SPLINE
SPL {X  -134.058, Y  +288.094, Z    +0.000, E1   +46.503, E3 +198295.093}
SPL {X  -148.633, Y  +314.028, Z    +0.000, E1   +38.752, E3 +198303.982}
SPL {X  -156.325, Y  +334.971, Z    +0.000, E1   +30.037, E3 +198307.750}
SPL {X  -160.130, Y  +351.024, Z    +0.000, E1   +21.715, E3 +198311.064}
SPL {X  -162.127, Y  +365.491, Z    +0.000, E1   +12.692, E3 +198310.988}
SPL {X  -162.801, Y  +378.004, Z    +0.000, E1    +3.811, E3 +198311.404}
SPL {X  -162.820, Y  +382.501, Z    +0.000, E1    +0.028, E3 +198310.822}
SPL {X  -162.820, Y  +385.123, Z    +0.000, E1    -3.284, E3 +198310.499}
SPL {X  -162.820, Y  +390.608, Z    +0.000, E1   -12.198, E3 +198310.413}
SPL {X  -162.820, Y  +396.028, Z    +0.000, E1   -22.022, E3 +198310.281}
SPL {X  -162.820, Y  +402.037, Z    +0.000, E1   -32.247, E3 +198310.219}
SPL {X  -162.820, Y  +411.189, Z    +0.000, E1   -44.140, E3 +198311.548}
SPL {X  -162.820, Y  +422.160, Z    +0.000, E1   -56.042, E3 +198310.020}
SPL {X  -162.820, Y  +475.891, Z    +0.000, E1   -67.666, E3 +198330.339}
SPL {X  -162.820, Y  +573.811, Z    +0.000, E1   -65.269, E3 +198414.937}
SPL {X  -162.820, Y  +580.233, Z    +0.000, E1   -64.427, E3 +198427.644}
SPL {X  -162.820, Y  +590.756, Z    +0.000, E1   -64.410, E3 +198438.211}
SPL {X  -162.820, Y  +600.605, Z    +0.000, E1   -64.446, E3 +198447.785}
SPL {X  -162.820, Y  +611.699, Z    +0.000, E1   -64.369, E3 +198459.464}
SPL {X  -162.820, Y  +622.825, Z    +0.000, E1   -64.446, E3 +198469.909}
SPL {X  -162.820, Y  +635.776, Z    +0.000, E1   -64.495, E3 +198482.598}
SPL {X  -162.820, Y  +648.933, Z    +0.000, E1   -64.417, E3 +198496.145}
SPL {X  -162.820, Y  +658.800, Z    +0.000, E1   -64.418, E3 +198505.960}
SPL {X  -162.820, Y  +670.777, Z    +0.000, E1   -64.432, E3 +198517.873}
SPL {X  -162.296, Y  +686.556, Z    +0.000, E1   -64.388, E3 +198534.076}
SPL {X  -160.469, Y  +701.070, Z    +0.000, E1   -64.058, E3 +198550.979}
SPL {X  -157.811, Y  +713.575, Z    +0.000, E1   -63.758, E3 +198565.558}
SPL {X  -155.696, Y  +721.135, Z    +0.000, E1   -63.387, E3 +198575.491}
SPL {X  -153.915, Y  +726.609, Z    +0.000, E1   -63.196, E3 +198582.266}
SPL {X  -151.802, Y  +732.376, Z    +0.000, E1   -62.761, E3 +198590.807}
SPL {X  -149.758, Y  +737.398, Z    +0.000, E1   -62.434, E3 +198597.828}
SPL {X  -146.903, Y  +743.713, Z    +0.000, E1   -62.188, E3 +198605.600}
SPL {X  -143.515, Y  +750.401, Z    +0.000, E1   -61.484, E3 +198616.285}
SPL {X  -140.303, Y  +756.116, Z    +0.000, E1   -60.974, E3 +198624.482}
SPL {X  -137.988, Y  +759.927, Z    +0.000, E1   -60.537, E3 +198630.416}
SPL {X  -134.516, Y  +765.238, Z    +0.000, E1   -60.629, E3 +198635.219}
SPL {X  -126.113, Y  +776.485, Z    +0.000, E1   -62.672, E3 +198636.779}
SPL {X   -95.040, Y  +805.704, Z    +0.000, E1   -55.103, E3 +198727.739}
ENDSPLINE

SPLINE
SPL {X   -95.634, Y  +805.274, Z    +0.000, E1   -52.767, E3 +198766.898}
SPL {X  -130.051, Y  +771.465, Z    +0.000, E1   -46.832, E3 +198865.304}
SPL {X  -154.243, Y  +725.647, Z    +0.000, E1   -32.659, E3 +198886.866}
SPL {X  -160.324, Y  +701.901, Z    +0.000, E1   -20.534, E3 +198887.689}
SPL {X  -161.938, Y  +690.423, Z    +0.000, E1   -13.625, E3 +198889.080}
SPL {X  -162.746, Y  +678.392, Z    +0.000, E1    -5.513, E3 +198889.152}
SPL {X  -162.820, Y  +671.700, Z    +0.000, E1    -0.272, E3 +198888.718}
SPL {X  -162.820, Y  +668.888, Z    +0.000, E1    +3.063, E3 +198888.415}
SPL {X  -162.820, Y  +664.763, Z    +0.000, E1    +9.526, E3 +198888.075}
SPL {X  -162.820, Y  +660.761, Z    +0.000, E1   +16.102, E3 +198888.414}
SPL {X  -162.820, Y  +655.024, Z    +0.000, E1   +25.730, E3 +198888.575}
SPL {X  -162.820, Y  +646.498, Z    +0.000, E1   +39.738, E3 +198887.096}
SPL {X  -162.820, Y  +637.711, Z    +0.000, E1   +46.793, E3 +198891.589}
SPL {X  -162.820, Y  +598.602, Z    +0.000, E1   +67.541, E3 +198894.140}
SPL {X  -162.820, Y  +578.435, Z    +0.000, E1   +65.472, E3 +198912.240}
SPL {X  -162.820, Y  +475.450, Z    +0.000, E1   +67.130, E3 +198981.177}
ENDSPLINE

SPLINE
SPL {X  -162.820, Y  +483.223, Z    +0.000, E1   +64.312, E3 +198995.617}
SPL {X  -162.820, Y  +502.830, Z    +0.000, E1   +59.229, E3 +199010.538}
ENDSPLINE

SPLINE
SPL {X  -162.820, Y  +486.621, Z    +0.000, E1   +59.661, E3 +199027.457}
SPL {X  -162.820, Y  +472.771, Z    +0.000, E1   +60.369, E3 +199039.203}
SPL {X  -162.820, Y  +460.138, Z    +0.000, E1   +61.014, E3 +199049.522}
SPL {X  -162.820, Y  +448.741, Z    +0.000, E1   +61.510, E3 +199059.037}
SPL {X  -162.820, Y  +430.985, Z    +0.000, E1   +62.533, E3 +199071.470}
SPL {X  -162.820, Y  +413.005, Z    +0.000, E1   +63.234, E3 +199085.460}
SPL {X  -162.820, Y  +396.727, Z    +0.000, E1   +63.972, E3 +199096.811}
SPL {X  -162.756, Y  +375.937, Z    +0.000, E1   +64.914, E3 +199110.421}
SPL {X  -161.353, Y  +358.691, Z    +0.000, E1   +65.588, E3 +199121.645}
SPL {X  -158.833, Y  +344.688, Z    +0.000, E1   +65.800, E3 +199133.108}
SPL {X  -156.326, Y  +334.977, Z    +0.000, E1   +65.428, E3 +199144.581}
SPL {X  -153.776, Y  +326.991, Z    +0.000, E1   +65.023, E3 +199154.844}
SPL {X  -149.992, Y  +317.154, Z    +0.000, E1   +64.515, E3 +199167.308}
SPL {X  -146.026, Y  +308.480, Z    +0.000, E1   +63.813, E3 +199179.550}
SPL {X  -142.454, Y  +301.650, Z    +0.000, E1   +63.360, E3 +199188.314}
SPL {X  -139.696, Y  +296.861, Z    +0.000, E1   +62.910, E3 +199195.082}
SPL {X  -137.330, Y  +293.030, Z    +0.000, E1   +62.290, E3 +199201.706}
SPL {X  -134.245, Y  +288.366, Z    +0.000, E1   +62.031, E3 +199207.188}
SPL {X  -128.642, Y  +280.693, Z    +0.000, E1   +63.351, E3 +199208.181}
SPL {X   -90.696, Y  +245.280, Z    +0.000, E1   +54.124, E3 +199328.870}
ENDSPLINE

SPLINE
SPL {X  -134.058, Y  +288.094, Z    +0.000, E1   +46.503, E3 +199456.384}
SPL {X  -153.979, Y  +327.577, Z    +0.000, E1   +33.452, E3 +199467.924}
SPL {X  -160.130, Y  +351.024, Z    +0.000, E1   +21.715, E3 +199472.354}
SPL {X  -162.127, Y  +365.491, Z    +0.000, E1   +12.692, E3 +199472.278}
SPL {X  -162.801, Y  +378.004, Z    +0.000, E1    +3.811, E3 +199472.694}
SPL {X  -162.820, Y  +382.501, Z    +0.000, E1    +0.028, E3 +199472.112}
SPL {X  -162.820, Y  +385.123, Z    +0.000, E1    -3.284, E3 +199471.790}
SPL {X  -162.820, Y  +390.608, Z    +0.000, E1   -12.198, E3 +199471.703}
SPL {X  -162.820, Y  +396.028, Z    +0.000, E1   -22.022, E3 +199471.571}
SPL {X  -162.820, Y  +402.037, Z    +0.000, E1   -32.247, E3 +199471.509}
SPL {X  -162.820, Y  +414.067, Z    +0.000, E1   -47.235, E3 +199472.935}
SPL {X  -162.820, Y  +424.566, Z    +0.000, E1   -59.255, E3 +199469.600}
SPL {X  -162.820, Y  +460.664, Z    +0.000, E1   -69.605, E3 +199477.896}
SPL {X  -162.820, Y  +481.040, Z    +0.000, E1   -67.047, E3 +199496.485}
SPL {X  -162.820, Y  +576.352, Z    +0.000, E1   -67.140, E3 +199564.004}
ENDSPLINE

SPLINE
SPL {X  -162.820, Y  +573.336, Z    +0.000, E1   -64.995, E3 +199577.756}
ENDSPLINE

SPLINE
SPL {X  -162.820, Y  +580.233, Z    +0.000, E1   -64.427, E3 +199588.934}
SPL {X  -162.820, Y  +590.756, Z    +0.000, E1   -64.410, E3 +199599.502}
SPL {X  -162.820, Y  +600.605, Z    +0.000, E1   -64.446, E3 +199609.075}
SPL {X  -162.820, Y  +611.699, Z    +0.000, E1   -64.369, E3 +199620.754}
SPL {X  -162.820, Y  +622.825, Z    +0.000, E1   -64.446, E3 +199631.199}
SPL {X  -162.820, Y  +635.776, Z    +0.000, E1   -64.495, E3 +199643.889}
SPL {X  -162.820, Y  +648.933, Z    +0.000, E1   -64.417, E3 +199657.436}
SPL {X  -162.820, Y  +658.800, Z    +0.000, E1   -64.418, E3 +199667.250}
SPL {X  -162.820, Y  +670.777, Z    +0.000, E1   -64.432, E3 +199679.163}
SPL {X  -162.296, Y  +686.556, Z    +0.000, E1   -64.388, E3 +199695.366}
SPL {X  -160.469, Y  +701.070, Z    +0.000, E1   -64.058, E3 +199712.269}
SPL {X  -157.811, Y  +713.575, Z    +0.000, E1   -63.758, E3 +199726.848}
SPL {X  -154.601, Y  +724.576, Z    +0.000, E1   -63.303, E3 +199740.970}
SPL {X  -151.802, Y  +732.376, Z    +0.000, E1   -62.761, E3 +199752.097}
SPL {X  -149.758, Y  +737.398, Z    +0.000, E1   -62.434, E3 +199759.118}
SPL {X  -146.903, Y  +743.713, Z    +0.000, E1   -62.188, E3 +199766.891}
SPL {X  -143.515, Y  +750.401, Z    +0.000, E1   -61.484, E3 +199777.575}
SPL {X  -138.985, Y  +758.314, Z    +0.000, E1   -60.770, E3 +199789.134}
SPL {X  -133.449, Y  +766.783, Z    +0.000, E1   -60.899, E3 +199796.754}
SPL {X   -94.739, Y  +805.919, Z    +0.000, E1   -54.063, E3 +199904.811}
ENDSPLINE

SPLINE
SPL {X  -130.051, Y  +771.465, Z    +0.000, E1   -46.832, E3 +200026.595}
SPL {X  -154.243, Y  +725.647, Z    +0.000, E1   -32.659, E3 +200048.157}
SPL {X  -160.324, Y  +701.901, Z    +0.000, E1   -20.534, E3 +200048.980}
SPL {X  -161.938, Y  +690.423, Z    +0.000, E1   -13.625, E3 +200050.370}
SPL {X  -162.638, Y  +681.194, Z    +0.000, E1    -7.430, E3 +200050.191}
SPL {X  -162.820, Y  +672.793, Z    +0.000, E1    -1.263, E3 +200050.249}
SPL {X  -162.820, Y  +670.674, Z    +0.000, E1    +0.808, E3 +200049.779}
SPL {X  -162.820, Y  +666.307, Z    +0.000, E1    +6.851, E3 +200049.562}
SPL {X  -162.820, Y  +660.761, Z    +0.000, E1   +16.102, E3 +200049.705}
SPL {X  -162.820, Y  +655.024, Z    +0.000, E1   +25.730, E3 +200049.866}
SPL {X  -162.820, Y  +646.498, Z    +0.000, E1   +39.738, E3 +200048.387}
SPL {X  -162.820, Y  +637.711, Z    +0.000, E1   +46.793, E3 +200052.879}
SPL {X  -162.820, Y  +598.602, Z    +0.000, E1   +67.541, E3 +200055.430}
SPL {X  -162.820, Y  +578.435, Z    +0.000, E1   +65.472, E3 +200073.530}
SPL {X  -162.820, Y  +480.401, Z    +0.000, E1   +65.660, E3 +200149.459}
ENDSPLINE

SPLINE
SPL {X  -162.820, Y  +490.253, Z    +0.000, E1   +62.754, E3 +200161.222}
SPL {X  -162.820, Y  +503.236, Z    +0.000, E1   +58.858, E3 +200173.575}
ENDSPLINE

SPLINE
SPL {X  -162.820, Y  +486.621, Z    +0.000, E1   +59.661, E3 +200188.748}
SPL {X  -162.820, Y  +472.771, Z    +0.000, E1   +60.369, E3 +200200.493}
SPL {X  -162.820, Y  +460.138, Z    +0.000, E1   +61.014, E3 +200210.813}
SPL {X  -162.820, Y  +448.741, Z    +0.000, E1   +61.510, E3 +200220.327}
SPL {X  -162.820, Y  +430.985, Z    +0.000, E1   +62.533, E3 +200232.760}
SPL {X  -162.820, Y  +413.005, Z    +0.000, E1   +63.234, E3 +200246.750}
SPL {X  -162.820, Y  +396.727, Z    +0.000, E1   +63.972, E3 +200258.102}
SPL {X  -162.756, Y  +375.937, Z    +0.000, E1   +64.914, E3 +200271.711}
SPL {X  -161.353, Y  +358.691, Z    +0.000, E1   +65.588, E3 +200282.936}
SPL {X  -159.475, Y  +347.667, Z    +0.000, E1   +65.889, E3 +200290.816}
SPL {X  -157.043, Y  +337.513, Z    +0.000, E1   +65.541, E3 +200302.894}
SPL {X  -154.736, Y  +329.832, Z    +0.000, E1   +65.034, E3 +200313.340}
SPL {X  -151.631, Y  +321.184, Z    +0.000, E1   +64.776, E3 +200323.185}
SPL {X  -147.832, Y  +312.265, Z    +0.000, E1   +64.201, E3 +200334.994}
SPL {X  -145.264, Y  +306.955, Z    +0.000, E1   +63.555, E3 +200343.600}
SPL {X  -142.454, Y  +301.650, Z    +0.000, E1   +63.360, E3 +200349.604}
SPL {X  -139.696, Y  +296.861, Z    +0.000, E1   +62.910, E3 +200356.372}
SPL {X  -137.330, Y  +293.030, Z    +0.000, E1   +62.290, E3 +200362.997}
SPL {X  -134.245, Y  +288.366, Z    +0.000, E1   +62.031, E3 +200368.478}
SPL {X  -128.642, Y  +280.693, Z    +0.000, E1   +63.351, E3 +200369.472}
SPL {X   -90.696, Y  +245.280, Z    +0.000, E1   +54.124, E3 +200490.160}
ENDSPLINE

SPLINE
SPL {X  -134.058, Y  +288.094, Z    +0.000, E1   +46.503, E3 +200617.674}
SPL {X  -153.979, Y  +327.577, Z    +0.000, E1   +33.452, E3 +200629.214}
SPL {X  -160.130, Y  +351.024, Z    +0.000, E1   +21.715, E3 +200633.645}
SPL {X  -162.127, Y  +365.491, Z    +0.000, E1   +12.692, E3 +200633.568}
SPL {X  -162.745, Y  +375.564, Z    +0.000, E1    +5.577, E3 +200634.179}
SPL {X  -162.820, Y  +382.222, Z    +0.000, E1    +0.380, E3 +200633.451}
SPL {X  -162.820, Y  +384.010, Z    +0.000, E1    -1.878, E3 +200633.114}
SPL {X  -162.820, Y  +387.631, Z    +0.000, E1    -7.169, E3 +200633.067}
SPL {X  -162.820, Y  +394.064, Z    +0.000, E1   -18.298, E3 +200632.878}
SPL {X  -162.820, Y  +402.037, Z    +0.000, E1   -32.247, E3 +200632.799}
SPL {X  -162.820, Y  +411.189, Z    +0.000, E1   -44.140, E3 +200634.129}
SPL {X  -162.820, Y  +422.160, Z    +0.000, E1   -56.042, E3 +200632.601}
SPL {X  -162.820, Y  +475.891, Z    +0.000, E1   -67.666, E3 +200652.919}
SPL {X  -162.820, Y  +573.811, Z    +0.000, E1   -65.269, E3 +200737.518}
SPL {X  -162.820, Y  +580.233, Z    +0.000, E1   -64.427, E3 +200750.224}
SPL {X  -162.820, Y  +590.756, Z    +0.000, E1   -64.410, E3 +200760.792}
SPL {X  -162.820, Y  +600.605, Z    +0.000, E1   -64.446, E3 +200770.365}
SPL {X  -162.820, Y  +611.699, Z    +0.000, E1   -64.369, E3 +200782.045}
SPL {X  -162.820, Y  +622.825, Z    +0.000, E1   -64.446, E3 +200792.489}
SPL {X  -162.820, Y  +635.776, Z    +0.000, E1   -64.495, E3 +200805.179}
SPL {X  -162.820, Y  +648.933, Z    +0.000, E1   -64.417, E3 +200818.726}
SPL {X  -162.820, Y  +658.800, Z    +0.000, E1   -64.418, E3 +200828.540}
SPL {X  -162.820, Y  +670.777, Z    +0.000, E1   -64.432, E3 +200840.453}
SPL {X  -162.296, Y  +686.556, Z    +0.000, E1   -64.388, E3 +200856.657}
SPL {X  -160.469, Y  +701.070, Z    +0.000, E1   -64.058, E3 +200873.560}
SPL {X  -157.811, Y  +713.575, Z    +0.000, E1   -63.758, E3 +200888.138}
SPL {X  -155.696, Y  +721.135, Z    +0.000, E1   -63.387, E3 +200898.072}
SPL {X  -153.915, Y  +726.609, Z    +0.000, E1   -63.196, E3 +200904.846}
SPL {X  -151.802, Y  +732.376, Z    +0.000, E1   -62.761, E3 +200913.388}
SPL {X  -149.758, Y  +737.398, Z    +0.000, E1   -62.434, E3 +200920.408}
SPL {X  -146.903, Y  +743.713, Z    +0.000, E1   -62.188, E3 +200928.181}
SPL {X  -144.901, Y  +747.758, Z    +0.000, E1   -61.566, E3 +200935.644}
SPL {X  -141.375, Y  +754.268, Z    +0.000, E1   -61.208, E3 +200944.198}
SPL {X  -137.124, Y  +761.291, Z    +0.000, E1   -60.398, E3 +200955.109}
SPL {X  -130.896, Y  +770.333, Z    +0.000, E1   -61.755, E3 +200957.784}
SPL {X   -94.739, Y  +805.919, Z    +0.000, E1   -54.063, E3 +201066.101}
ENDSPLINE

SPLINE
SPL {X  -130.051, Y  +771.465, Z    +0.000, E1   -46.832, E3 +201187.885}
SPL {X  -150.288, Y  +736.141, Z    +0.000, E1   -36.889, E3 +201207.741}
SPL {X  -159.122, Y  +708.003, Z    +0.000, E1   -24.018, E3 +201210.449}
SPL {X  -161.938, Y  +690.423, Z    +0.000, E1   -13.625, E3 +201211.660}
SPL {X  -162.746, Y  +678.392, Z    +0.000, E1    -5.513, E3 +201211.733}
SPL {X  -162.820, Y  +671.700, Z    +0.000, E1    -0.272, E3 +201211.299}
SPL {X  -162.820, Y  +668.888, Z    +0.000, E1    +3.063, E3 +201210.996}
SPL {X  -162.820, Y  +664.763, Z    +0.000, E1    +9.526, E3 +201210.655}
SPL {X  -162.820, Y  +660.761, Z    +0.000, E1   +16.102, E3 +201210.995}
SPL {X  -162.820, Y  +655.024, Z    +0.000, E1   +25.730, E3 +201211.156}
SPL {X  -162.820, Y  +646.498, Z    +0.000, E1   +39.738, E3 +201209.677}
SPL {X  -162.820, Y  +637.711, Z    +0.000, E1   +46.793, E3 +201214.170}
SPL {X  -162.820, Y  +613.264, Z    +0.000, E1   +68.325, E3 +201206.368}
SPL {X  -162.820, Y  +583.199, Z    +0.000, E1   +66.160, E3 +201229.858}
SPL {X  -162.820, Y  +480.401, Z    +0.000, E1   +65.660, E3 +201310.749}
ENDSPLINE

SPLINE
SPL {X  -162.820, Y  +490.253, Z    +0.000, E1   +62.754, E3 +201322.512}
SPL {X  -162.820, Y  +503.236, Z    +0.000, E1   +58.858, E3 +201334.866}
ENDSPLINE

SPLINE
SPL {X  -162.820, Y  +486.621, Z    +0.000, E1   +59.661, E3 +201350.038}
SPL {X  -162.820, Y  +472.771, Z    +0.000, E1   +60.369, E3 +201361.783}
SPL {X  -162.820, Y  +460.138, Z    +0.000, E1   +61.014, E3 +201372.103}
SPL {X  -162.820, Y  +448.741, Z    +0.000, E1   +61.510, E3 +201381.618}
SPL {X  -162.820, Y  +430.985, Z    +0.000, E1   +62.533, E3 +201394.051}
SPL {X  -162.820, Y  +413.005, Z    +0.000, E1   +63.234, E3 +201408.041}
SPL {X  -162.820, Y  +396.727, Z    +0.000, E1   +63.972, E3 +201419.392}
SPL {X  -162.756, Y  +375.937, Z    +0.000, E1   +64.914, E3 +201433.001}
SPL {X  -161.353, Y  +358.691, Z    +0.000, E1   +65.588, E3 +201444.226}
SPL {X  -159.475, Y  +347.667, Z    +0.000, E1   +65.889, E3 +201452.107}
SPL {X  -157.043, Y  +337.513, Z    +0.000, E1   +65.541, E3 +201464.184}
SPL {X  -153.776, Y  +326.991, Z    +0.000, E1   +65.023, E3 +201477.425}
SPL {X  -149.992, Y  +317.154, Z    +0.000, E1   +64.515, E3 +201489.889}
SPL {X  -146.026, Y  +308.480, Z    +0.000, E1   +63.813, E3 +201502.131}
SPL {X  -142.454, Y  +301.650, Z    +0.000, E1   +63.360, E3 +201510.894}
SPL {X  -139.696, Y  +296.861, Z    +0.000, E1   +62.910, E3 +201517.662}
SPL {X  -137.330, Y  +293.030, Z    +0.000, E1   +62.290, E3 +201524.287}
SPL {X  -134.245, Y  +288.366, Z    +0.000, E1   +62.031, E3 +201529.769}
SPL {X  -128.642, Y  +280.693, Z    +0.000, E1   +63.351, E3 +201530.762}
SPL {X   -90.696, Y  +245.280, Z    +0.000, E1   +54.124, E3 +201651.451}
ENDSPLINE

SPLINE
SPL {X  -134.058, Y  +288.094, Z    +0.000, E1   +46.503, E3 +201778.964}
SPL {X  -153.979, Y  +327.577, Z    +0.000, E1   +33.452, E3 +201790.504}
SPL {X  -160.130, Y  +351.024, Z    +0.000, E1   +21.715, E3 +201794.935}
SPL {X  -162.127, Y  +365.491, Z    +0.000, E1   +12.692, E3 +201794.859}
SPL {X  -162.745, Y  +375.564, Z    +0.000, E1    +5.577, E3 +201795.469}
SPL {X  -162.820, Y  +382.222, Z    +0.000, E1    +0.380, E3 +201794.742}
SPL {X  -162.820, Y  +385.123, Z    +0.000, E1    -3.284, E3 +201794.370}
SPL {X  -162.820, Y  +390.608, Z    +0.000, E1   -12.198, E3 +201794.284}
SPL {X  -162.820, Y  +396.028, Z    +0.000, E1   -22.022, E3 +201794.152}
SPL {X  -162.820, Y  +402.037, Z    +0.000, E1   -32.247, E3 +201794.090}
SPL {X  -162.820, Y  +411.189, Z    +0.000, E1   -44.140, E3 +201795.419}
SPL {X  -162.820, Y  +422.160, Z    +0.000, E1   -56.042, E3 +201793.891}
SPL {X  -162.820, Y  +475.891, Z    +0.000, E1   -67.666, E3 +201814.210}
SPL {X  -162.820, Y  +573.811, Z    +0.000, E1   -65.269, E3 +201898.808}
SPL {X  -162.820, Y  +580.233, Z    +0.000, E1   -64.427, E3 +201911.515}
SPL {X  -162.820, Y  +590.756, Z    +0.000, E1   -64.410, E3 +201922.082}
SPL {X  -162.820, Y  +600.605, Z    +0.000, E1   -64.446, E3 +201931.656}
SPL {X  -162.820, Y  +611.699, Z    +0.000, E1   -64.369, E3 +201943.335}
SPL {X  -162.820, Y  +622.825, Z    +0.000, E1   -64.446, E3 +201953.780}
SPL {X  -162.820, Y  +635.776, Z    +0.000, E1   -64.495, E3 +201966.469}
SPL {X  -162.820, Y  +648.933, Z    +0.000, E1   -64.417, E3 +201980.016}
SPL {X  -162.820, Y  +658.800, Z    +0.000, E1   -64.418, E3 +201989.831}
SPL {X  -162.820, Y  +670.777, Z    +0.000, E1   -64.432, E3 +202001.744}
SPL {X  -162.296, Y  +686.556, Z    +0.000, E1   -64.388, E3 +202017.947}
SPL {X  -160.469, Y  +701.070, Z    +0.000, E1   -64.058, E3 +202034.850}
SPL {X  -157.811, Y  +713.575, Z    +0.000, E1   -63.758, E3 +202049.429}
SPL {X  -155.696, Y  +721.135, Z    +0.000, E1   -63.387, E3 +202059.362}
SPL {X  -153.915, Y  +726.609, Z    +0.000, E1   -63.196, E3 +202066.137}
SPL {X  -151.802, Y  +732.376, Z    +0.000, E1   -62.761, E3 +202074.678}
SPL {X  -149.758, Y  +737.398, Z    +0.000, E1   -62.434, E3 +202081.699}
SPL {X  -146.903, Y  +743.713, Z    +0.000, E1   -62.188, E3 +202089.471}
SPL {X  -143.515, Y  +750.401, Z    +0.000, E1   -61.484, E3 +202100.156}
SPL {X  -140.303, Y  +756.116, Z    +0.000, E1   -60.974, E3 +202108.353}
SPL {X  -137.124, Y  +761.291, Z    +0.000, E1   -60.398, E3 +202116.400}
SPL {X  -130.896, Y  +770.333, Z    +0.000, E1   -61.755, E3 +202119.074}
SPL {X   -94.739, Y  +805.919, Z    +0.000, E1   -54.063, E3 +202227.391}
ENDSPLINE

SPLINE
SPL {X  -130.051, Y  +771.465, Z    +0.000, E1   -46.832, E3 +202349.175}
SPL {X  -154.243, Y  +725.647, Z    +0.000, E1   -32.659, E3 +202370.737}
SPL {X  -161.394, Y  +695.005, Z    +0.000, E1   -16.571, E3 +202372.442}
SPL {X  -162.746, Y  +678.392, Z    +0.000, E1    -5.513, E3 +202373.023}
SPL {X  -162.820, Y  +672.097, Z    +0.000, E1    -0.584, E3 +202372.728}
SPL {X  -162.820, Y  +671.335, Z    +0.000, E1    +0.161, E3 +202372.461}
SPL {X  -162.820, Y  +668.888, Z    +0.000, E1    +3.063, E3 +202372.286}
SPL {X  -162.820, Y  +664.763, Z    +0.000, E1    +9.526, E3 +202371.946}
SPL {X  -162.820, Y  +660.761, Z    +0.000, E1   +16.102, E3 +202372.285}
SPL {X  -162.820, Y  +655.024, Z    +0.000, E1   +25.730, E3 +202372.446}
SPL {X  -162.820, Y  +646.498, Z    +0.000, E1   +39.738, E3 +202370.967}
SPL {X  -162.820, Y  +637.711, Z    +0.000, E1   +46.793, E3 +202375.460}
SPL {X  -162.820, Y  +598.602, Z    +0.000, E1   +67.541, E3 +202378.011}
SPL {X  -162.820, Y  +578.435, Z    +0.000, E1   +65.472, E3 +202396.111}
SPL {X  -162.820, Y  +480.401, Z    +0.000, E1   +65.660, E3 +202472.040}
ENDSPLINE

SPLINE
SPL {X  -162.820, Y  +490.253, Z    +0.000, E1   +62.754, E3 +202483.802}
SPL {X  -162.820, Y  +503.236, Z    +0.000, E1   +58.858, E3 +202496.156}
ENDSPLINE

SPLINE
SPL {X  -162.820, Y  +486.621, Z    +0.000, E1   +59.661, E3 +202511.328}
SPL {X  -162.820, Y  +472.771, Z    +0.000, E1   +60.369, E3 +202523.074}
SPL {X  -162.820, Y  +460.138, Z    +0.000, E1   +61.014, E3 +202533.393}
SPL {X  -162.820, Y  +442.137, Z    +0.000, E1   +61.946, E3 +202547.290}
SPL {X  -162.820, Y  +425.982, Z    +0.000, E1   +62.713, E3 +202559.316}
SPL {X  -162.820, Y  +413.005, Z    +0.000, E1   +63.234, E3 +202569.331}
SPL {X  -162.820, Y  +396.727, Z    +0.000, E1   +63.972, E3 +202580.682}
SPL {X  -162.820, Y  +382.966, Z    +0.000, E1   +64.511, E3 +202590.405}
SPL {X  -161.867, Y  +362.911, Z    +0.000, E1   +65.480, E3 +202602.478}
SPL {X  -158.833, Y  +344.688, Z    +0.000, E1   +65.800, E3 +202616.979}
SPL {X  -156.326, Y  +334.977, Z    +0.000, E1   +65.428, E3 +202628.452}
SPL {X  -153.776, Y  +326.991, Z    +0.000, E1   +65.023, E3 +202638.715}
SPL {X  -150.991, Y  +319.573, Z    +0.000, E1   +64.614, E3 +202648.169}
SPL {X  -147.832, Y  +312.265, Z    +0.000, E1   +64.201, E3 +202657.575}
SPL {X  -145.264, Y  +306.955, Z    +0.000, E1   +63.555, E3 +202666.181}
SPL {X  -142.454, Y  +301.650, Z    +0.000, E1   +63.360, E3 +202672.185}
SPL {X  -139.696, Y  +296.861, Z    +0.000, E1   +62.910, E3 +202678.953}
SPL {X  -137.330, Y  +293.030, Z    +0.000, E1   +62.290, E3 +202685.577}
SPL {X  -134.245, Y  +288.366, Z    +0.000, E1   +62.031, E3 +202691.059}
SPL {X  -128.642, Y  +280.693, Z    +0.000, E1   +63.351, E3 +202692.052}
SPL {X   -90.696, Y  +245.280, Z    +0.000, E1   +54.124, E3 +202812.741}
ENDSPLINE

SPLINE
SPL {X  -134.058, Y  +288.094, Z    +0.000, E1   +46.503, E3 +202940.255}
SPL {X  -148.633, Y  +314.028, Z    +0.000, E1   +38.752, E3 +202949.143}
SPL {X  -156.325, Y  +334.971, Z    +0.000, E1   +30.037, E3 +202952.911}
SPL {X  -160.130, Y  +351.024, Z    +0.000, E1   +21.715, E3 +202956.225}
SPL {X  -162.127, Y  +365.491, Z    +0.000, E1   +12.692, E3 +202956.149}
SPL {X  -162.801, Y  +378.004, Z    +0.000, E1    +3.811, E3 +202956.565}
SPL {X  -162.820, Y  +382.501, Z    +0.000, E1    +0.028, E3 +202955.983}
SPL {X  -162.820, Y  +384.010, Z    +0.000, E1    -1.878, E3 +202955.694}
SPL {X  -162.820, Y  +387.631, Z    +0.000, E1    -7.169, E3 +202955.648}
SPL {X  -162.820, Y  +394.064, Z    +0.000, E1   -18.298, E3 +202955.458}
SPL {X  -162.820, Y  +402.037, Z    +0.000, E1   -32.247, E3 +202955.380}
SPL {X  -162.820, Y  +411.189, Z    +0.000, E1   -44.140, E3 +202956.710}
SPL {X  -162.820, Y  +422.160, Z    +0.000, E1   -56.042, E3 +202955.181}
SPL {X  -162.820, Y  +475.891, Z    +0.000, E1   -67.666, E3 +202975.500}
SPL {X  -162.820, Y  +573.811, Z    +0.000, E1   -65.269, E3 +203060.098}
SPL {X  -162.820, Y  +580.233, Z    +0.000, E1   -64.427, E3 +203072.805}
SPL {X  -162.820, Y  +590.756, Z    +0.000, E1   -64.410, E3 +203083.373}
SPL {X  -162.820, Y  +600.605, Z    +0.000, E1   -64.446, E3 +203092.946}
SPL {X  -162.820, Y  +611.699, Z    +0.000, E1   -64.369, E3 +203104.625}
SPL {X  -162.820, Y  +622.825, Z    +0.000, E1   -64.446, E3 +203115.070}
SPL {X  -162.820, Y  +635.776, Z    +0.000, E1   -64.495, E3 +203127.760}
SPL {X  -162.820, Y  +648.933, Z    +0.000, E1   -64.417, E3 +203141.307}
SPL {X  -162.820, Y  +658.800, Z    +0.000, E1   -64.418, E3 +203151.121}
SPL {X  -162.820, Y  +670.777, Z    +0.000, E1   -64.432, E3 +203163.034}
SPL {X  -162.613, Y  +681.710, Z    +0.000, E1   -64.310, E3 +203174.798}
SPL {X  -161.587, Y  +693.503, Z    +0.000, E1   -64.259, E3 +203187.152}
SPL {X  -159.311, Y  +707.123, Z    +0.000, E1   -64.022, E3 +203202.396}
SPL {X  -156.625, Y  +717.984, Z    +0.000, E1   -63.524, E3 +203216.751}
SPL {X  -153.915, Y  +726.609, Z    +0.000, E1   -63.196, E3 +203227.427}
SPL {X  -151.802, Y  +732.376, Z    +0.000, E1   -62.761, E3 +203235.968}
SPL {X  -149.758, Y  +737.398, Z    +0.000, E1   -62.434, E3 +203242.989}
SPL {X  -146.903, Y  +743.713, Z    +0.000, E1   -62.188, E3 +203250.762}
SPL {X  -143.515, Y  +750.401, Z    +0.000, E1   -61.484, E3 +203261.446}
SPL {X  -138.985, Y  +758.314, Z    +0.000, E1   -60.770, E3 +203273.005}
SPL {X  -133.449, Y  +766.783, Z    +0.000, E1   -60.899, E3 +203280.625}
SPL {X   -94.739, Y  +805.919, Z    +0.000, E1   -54.063, E3 +203388.682}
ENDSPLINE

SPLINE
SPL {X  -130.051, Y  +771.465, Z    +0.000, E1   -46.832, E3 +203510.466}
SPL {X  -154.243, Y  +725.647, Z    +0.000, E1   -32.659, E3 +203532.028}
SPL {X  -160.324, Y  +701.901, Z    +0.000, E1   -20.534, E3 +203532.851}
SPL {X  -161.938, Y  +690.423, Z    +0.000, E1   -13.625, E3 +203534.241}
SPL {X  -162.638, Y  +681.194, Z    +0.000, E1    -7.430, E3 +203534.062}
SPL {X  -162.820, Y  +672.793, Z    +0.000, E1    -1.263, E3 +203534.120}
SPL {X  -162.820, Y  +670.674, Z    +0.000, E1    +0.808, E3 +203533.650}
SPL {X  -162.820, Y  +666.307, Z    +0.000, E1    +6.851, E3 +203533.433}
SPL {X  -162.820, Y  +660.761, Z    +0.000, E1   +16.102, E3 +203533.576}
SPL {X  -162.820, Y  +655.024, Z    +0.000, E1   +25.730, E3 +203533.737}
SPL {X  -162.820, Y  +646.498, Z    +0.000, E1   +39.738, E3 +203532.258}
SPL {X  -162.820, Y  +637.711, Z    +0.000, E1   +46.793, E3 +203536.750}
SPL {X  -162.820, Y  +598.602, Z    +0.000, E1   +67.541, E3 +203539.301}
SPL {X  -162.820, Y  +578.435, Z    +0.000, E1   +65.472, E3 +203557.401}
SPL {X  -162.820, Y  +480.401, Z    +0.000, E1   +65.660, E3 +203633.330}
ENDSPLINE

SPLINE
SPL {X  -162.820, Y  +490.253, Z    +0.000, E1   +62.754, E3 +203645.093}
SPL {X  -162.820, Y  +503.236, Z    +0.000, E1   +58.858, E3 +203657.446}
ENDSPLINE

SPLINE
SPL {X  -162.820, Y  +486.621, Z    +0.000, E1   +59.661, E3 +203672.619}
SPL {X  -162.820, Y  +472.771, Z    +0.000, E1   +60.369, E3 +203684.364}
SPL {X  -162.820, Y  +460.138, Z    +0.000, E1   +61.014, E3 +203694.684}
SPL {X  -162.820, Y  +448.741, Z    +0.000, E1   +61.510, E3 +203704.198}
SPL {X  -162.820, Y  +430.985, Z    +0.000, E1   +62.533, E3 +203716.631}
SPL {X  -162.820, Y  +413.005, Z    +0.000, E1   +63.234, E3 +203730.621}
SPL {X  -162.820, Y  +396.727, Z    +0.000, E1   +63.972, E3 +203741.973}
SPL {X  -162.756, Y  +375.937, Z    +0.000, E1   +64.914, E3 +203755.582}
SPL {X  -161.353, Y  +358.691, Z    +0.000, E1   +65.588, E3 +203766.807}
SPL {X  -159.475, Y  +347.667, Z    +0.000, E1   +65.889, E3 +203774.687}
SPL {X  -157.043, Y  +337.513, Z    +0.000, E1   +65.541, E3 +203786.765}
SPL {X  -154.736, Y  +329.832, Z    +0.000, E1   +65.034, E3 +203797.211}
SPL {X  -151.631, Y  +321.184, Z    +0.000, E1   +64.776, E3 +203807.056}
SPL {X  -147.832, Y  +312.265, Z    +0.000, E1   +64.201, E3 +203818.865}
SPL {X  -145.264, Y  +306.955, Z    +0.000, E1   +63.555, E3 +203827.471}
SPL {X  -142.454, Y  +301.650, Z    +0.000, E1   +63.360, E3 +203833.475}
SPL {X  -139.696, Y  +296.861, Z    +0.000, E1   +62.910, E3 +203840.243}
SPL {X  -137.330, Y  +293.030, Z    +0.000, E1   +62.290, E3 +203846.868}
SPL {X  -134.245, Y  +288.366, Z    +0.000, E1   +62.031, E3 +203852.349}
SPL {X  -128.642, Y  +280.693, Z    +0.000, E1   +63.351, E3 +203853.343}
SPL {X   -90.696, Y  +245.280, Z    +0.000, E1   +54.124, E3 +203974.031}
ENDSPLINE

SPLINE
SPL {X  -134.058, Y  +288.094, Z    +0.000, E1   +46.503, E3 +204101.545}
SPL {X  -153.979, Y  +327.577, Z    +0.000, E1   +33.452, E3 +204113.085}
SPL {X  -160.130, Y  +351.024, Z    +0.000, E1   +21.715, E3 +204117.516}
SPL {X  -162.127, Y  +365.491, Z    +0.000, E1   +12.692, E3 +204117.439}
SPL {X  -162.745, Y  +375.564, Z    +0.000, E1    +5.577, E3 +204118.049}
SPL {X  -162.820, Y  +382.222, Z    +0.000, E1    +0.380, E3 +204117.322}
SPL {X  -162.820, Y  +384.010, Z    +0.000, E1    -1.878, E3 +204116.985}
SPL {X  -162.820, Y  +387.631, Z    +0.000, E1    -7.169, E3 +204116.938}
SPL {X  -162.820, Y  +394.064, Z    +0.000, E1   -18.298, E3 +204116.748}
SPL {X  -162.820, Y  +402.037, Z    +0.000, E1   -32.247, E3 +204116.670}
SPL {X  -162.820, Y  +411.189, Z    +0.000, E1   -44.140, E3 +204118.000}
SPL {X  -162.820, Y  +422.160, Z    +0.000, E1   -56.042, E3 +204116.472}
SPL {X  -162.820, Y  +475.891, Z    +0.000, E1   -67.666, E3 +204136.790}
SPL {X  -162.820, Y  +573.811, Z    +0.000, E1   -65.269, E3 +204221.389}
SPL {X  -162.820, Y  +580.233, Z    +0.000, E1   -64.427, E3 +204234.095}
SPL {X  -162.820, Y  +590.756, Z    +0.000, E1   -64.410, E3 +204244.663}
SPL {X  -162.820, Y  +600.605, Z    +0.000, E1   -64.446, E3 +204254.236}
SPL {X  -162.820, Y  +611.699, Z    +0.000, E1   -64.369, E3 +204265.916}
SPL {X  -162.820, Y  +622.825, Z    +0.000, E1   -64.446, E3 +204276.360}
SPL {X  -162.820, Y  +635.776, Z    +0.000, E1   -64.495, E3 +204289.050}
SPL {X  -162.820, Y  +648.933, Z    +0.000, E1   -64.417, E3 +204302.597}
SPL {X  -162.820, Y  +658.800, Z    +0.000, E1   -64.418, E3 +204312.411}
SPL {X  -162.820, Y  +670.777, Z    +0.000, E1   -64.432, E3 +204324.324}
SPL {X  -162.296, Y  +686.556, Z    +0.000, E1   -64.388, E3 +204340.528}
SPL {X  -160.469, Y  +701.070, Z    +0.000, E1   -64.058, E3 +204357.431}
SPL {X  -157.811, Y  +713.575, Z    +0.000, E1   -63.758, E3 +204372.009}
SPL {X  -155.696, Y  +721.135, Z    +0.000, E1   -63.387, E3 +204381.943}
SPL {X  -153.915, Y  +726.609, Z    +0.000, E1   -63.196, E3 +204388.717}
SPL {X  -151.802, Y  +732.376, Z    +0.000, E1   -62.761, E3 +204397.259}
SPL {X  -149.758, Y  +737.398, Z    +0.000, E1   -62.434, E3 +204404.279}
SPL {X  -146.903, Y  +743.713, Z    +0.000, E1   -62.188, E3 +204412.052}
SPL {X  -144.901, Y  +747.758, Z    +0.000, E1   -61.566, E3 +204419.515}
SPL {X  -141.375, Y  +754.268, Z    +0.000, E1   -61.208, E3 +204428.069}
SPL {X  -137.124, Y  +761.291, Z    +0.000, E1   -60.398, E3 +204438.980}
SPL {X  -130.896, Y  +770.333, Z    +0.000, E1   -61.755, E3 +204441.655}
SPL {X   -94.739, Y  +805.919, Z    +0.000, E1   -54.063, E3 +204549.972}
ENDSPLINE

SPLINE
SPL {X  -130.051, Y  +771.465, Z    +0.000, E1   -46.832, E3 +204671.756}
SPL {X  -150.288, Y  +736.141, Z    +0.000, E1   -36.889, E3 +204691.612}
SPL {X  -159.122, Y  +708.003, Z    +0.000, E1   -24.018, E3 +204694.320}
SPL {X  -161.938, Y  +690.423, Z    +0.000, E1   -13.625, E3 +204695.531}
SPL {X  -162.746, Y  +678.392, Z    +0.000, E1    -5.513, E3 +204695.604}
SPL {X  -162.820, Y  +671.700, Z    +0.000, E1    -0.272, E3 +204695.170}
SPL {X  -162.820, Y  +668.888, Z    +0.000, E1    +3.063, E3 +204694.867}
SPL {X  -162.820, Y  +664.763, Z    +0.000, E1    +9.526, E3 +204694.526}
SPL {X  -162.820, Y  +660.761, Z    +0.000, E1   +16.102, E3 +204694.866}
SPL {X  -162.820, Y  +655.024, Z    +0.000, E1   +25.730, E3 +204695.027}
SPL {X  -162.820, Y  +646.498, Z    +0.000, E1   +39.738, E3 +204693.548}
SPL {X  -162.820, Y  +637.711, Z    +0.000, E1   +46.793, E3 +204698.041}
SPL {X  -162.820, Y  +613.264, Z    +0.000, E1   +68.325, E3 +204690.239}
SPL {X  -162.820, Y  +583.199, Z    +0.000, E1   +66.160, E3 +204713.729}
SPL {X  -162.820, Y  +480.401, Z    +0.000, E1   +65.660, E3 +204794.620}
ENDSPLINE

SPLINE
SPL {X  -162.820, Y  +490.253, Z    +0.000, E1   +62.754, E3 +204806.383}
SPL {X  -162.820, Y  +503.236, Z    +0.000, E1   +58.858, E3 +204818.737}
ENDSPLINE

SPLINE
SPL {X  -162.820, Y  +486.621, Z    +0.000, E1   +59.661, E3 +204833.909}
SPL {X  -162.820, Y  +472.771, Z    +0.000, E1   +60.369, E3 +204845.654}
SPL {X  -162.820, Y  +460.138, Z    +0.000, E1   +61.014, E3 +204855.974}
SPL {X  -162.820, Y  +448.741, Z    +0.000, E1   +61.510, E3 +204865.489}
SPL {X  -162.820, Y  +430.985, Z    +0.000, E1   +62.533, E3 +204877.922}
SPL {X  -162.820, Y  +413.005, Z    +0.000, E1   +63.234, E3 +204891.912}
SPL {X  -162.820, Y  +396.727, Z    +0.000, E1   +63.972, E3 +204903.263}
SPL {X  -162.756, Y  +375.937, Z    +0.000, E1   +64.914, E3 +204916.872}
SPL {X  -161.353, Y  +358.691, Z    +0.000, E1   +65.588, E3 +204928.097}
SPL {X  -159.475, Y  +347.667, Z    +0.000, E1   +65.889, E3 +204935.977}
SPL {X  -157.043, Y  +337.513, Z    +0.000, E1   +65.541, E3 +204948.055}
SPL {X  -153.776, Y  +326.991, Z    +0.000, E1   +65.023, E3 +204961.296}
SPL {X  -149.992, Y  +317.154, Z    +0.000, E1   +64.515, E3 +204973.760}
SPL {X  -146.026, Y  +308.480, Z    +0.000, E1   +63.813, E3 +204986.002}
SPL {X  -142.454, Y  +301.650, Z    +0.000, E1   +63.360, E3 +204994.765}
SPL {X  -139.696, Y  +296.861, Z    +0.000, E1   +62.910, E3 +205001.533}
SPL {X  -137.330, Y  +293.030, Z    +0.000, E1   +62.290, E3 +205008.158}
SPL {X  -134.245, Y  +288.366, Z    +0.000, E1   +62.031, E3 +205013.639}
SPL {X  -128.642, Y  +280.693, Z    +0.000, E1   +63.351, E3 +205014.633}
SPL {X   -90.696, Y  +245.280, Z    +0.000, E1   +54.124, E3 +205135.322}
ENDSPLINE

SPLINE
SPL {X  -134.058, Y  +288.094, Z    +0.000, E1   +46.503, E3 +205262.835}
SPL {X  -153.979, Y  +327.577, Z    +0.000, E1   +33.452, E3 +205274.375}
SPL {X  -160.130, Y  +351.024, Z    +0.000, E1   +21.715, E3 +205278.806}
SPL {X  -162.127, Y  +365.491, Z    +0.000, E1   +12.692, E3 +205278.730}
SPL {X  -162.745, Y  +375.564, Z    +0.000, E1    +5.577, E3 +205279.340}
SPL {X  -162.820, Y  +382.222, Z    +0.000, E1    +0.380, E3 +205278.613}
SPL {X  -162.820, Y  +385.123, Z    +0.000, E1    -3.284, E3 +205278.241}
SPL {X  -162.820, Y  +390.608, Z    +0.000, E1   -12.198, E3 +205278.155}
SPL {X  -162.820, Y  +396.028, Z    +0.000, E1   -22.022, E3 +205278.023}
SPL {X  -162.820, Y  +402.037, Z    +0.000, E1   -32.247, E3 +205277.961}
SPL {X  -162.820, Y  +411.189, Z    +0.000, E1   -44.140, E3 +205279.290}
SPL {X  -162.820, Y  +422.160, Z    +0.000, E1   -56.042, E3 +205277.762}
SPL {X  -162.820, Y  +475.891, Z    +0.000, E1   -67.666, E3 +205298.081}
SPL {X  -162.820, Y  +576.352, Z    +0.000, E1   -67.140, E3 +205370.455}
ENDSPLINE

SPLINE
SPL {X  -162.820, Y  +573.336, Z    +0.000, E1   -64.995, E3 +205384.207}
ENDSPLINE

SPLINE
SPL {X  -162.820, Y  +580.233, Z    +0.000, E1   -64.427, E3 +205395.386}
SPL {X  -162.820, Y  +590.756, Z    +0.000, E1   -64.410, E3 +205405.953}
SPL {X  -162.820, Y  +600.605, Z    +0.000, E1   -64.446, E3 +205415.527}
SPL {X  -162.820, Y  +611.699, Z    +0.000, E1   -64.369, E3 +205427.206}
SPL {X  -162.820, Y  +622.825, Z    +0.000, E1   -64.446, E3 +205437.651}
SPL {X  -162.820, Y  +635.776, Z    +0.000, E1   -64.495, E3 +205450.340}
SPL {X  -162.820, Y  +648.933, Z    +0.000, E1   -64.417, E3 +205463.887}
SPL {X  -162.820, Y  +658.800, Z    +0.000, E1   -64.418, E3 +205473.701}
SPL {X  -162.820, Y  +670.777, Z    +0.000, E1   -64.432, E3 +205485.615}
SPL {X  -162.613, Y  +681.710, Z    +0.000, E1   -64.310, E3 +205497.379}
SPL {X  -161.587, Y  +693.503, Z    +0.000, E1   -64.259, E3 +205509.733}
SPL {X  -159.883, Y  +704.285, Z    +0.000, E1   -64.016, E3 +205522.073}
SPL {X  -157.811, Y  +713.575, Z    +0.000, E1   -63.758, E3 +205533.300}
SPL {X  -154.601, Y  +724.576, Z    +0.000, E1   -63.303, E3 +205547.422}
SPL {X  -151.802, Y  +732.376, Z    +0.000, E1   -62.761, E3 +205558.549}
SPL {X  -149.758, Y  +737.398, Z    +0.000, E1   -62.434, E3 +205565.570}
SPL {X  -146.903, Y  +743.713, Z    +0.000, E1   -62.188, E3 +205573.342}
SPL {X  -144.901, Y  +747.758, Z    +0.000, E1   -61.566, E3 +205580.805}
SPL {X  -141.375, Y  +754.268, Z    +0.000, E1   -61.208, E3 +205589.359}
SPL {X  -137.124, Y  +761.291, Z    +0.000, E1   -60.398, E3 +205600.271}
SPL {X  -130.896, Y  +770.333, Z    +0.000, E1   -61.755, E3 +205602.945}
SPL {X   -94.739, Y  +805.919, Z    +0.000, E1   -54.063, E3 +205711.262}
ENDSPLINE

SPLINE
SPL {X  -120.571, Y  +782.921, Z    +0.000, E1   -48.746, E3 +205818.559}
SPL {X  -145.902, Y  +745.770, Z    +0.000, E1   -40.275, E3 +205849.706}
SPL {X  -156.935, Y  +716.881, Z    +0.000, E1   -28.554, E3 +205855.695}
SPL {X  -161.394, Y  +695.005, Z    +0.000, E1   -16.571, E3 +205856.313}
SPL {X  -162.746, Y  +678.392, Z    +0.000, E1    -5.513, E3 +205856.894}
SPL {X  -162.820, Y  +671.700, Z    +0.000, E1    -0.272, E3 +205856.460}
SPL {X  -162.820, Y  +669.993, Z    +0.000, E1    +1.755, E3 +205856.126}
SPL {X  -162.820, Y  +666.307, Z    +0.000, E1    +6.851, E3 +205856.013}
SPL {X  -162.820, Y  +659.878, Z    +0.000, E1   +17.497, E3 +205856.221}
SPL {X  -162.820, Y  +650.308, Z    +0.000, E1   +33.487, E3 +205855.635}
SPL {X  -162.820, Y  +637.711, Z    +0.000, E1   +46.793, E3 +205859.331}
SPL {X  -162.820, Y  +613.264, Z    +0.000, E1   +68.325, E3 +205851.529}
SPL {X  -162.820, Y  +583.199, Z    +0.000, E1   +66.160, E3 +205875.019}
SPL {X  -162.820, Y  +480.401, Z    +0.000, E1   +65.660, E3 +205955.911}
ENDSPLINE

SPLINE
SPL {X  -162.820, Y  +490.253, Z    +0.000, E1   +62.754, E3 +205967.673}
SPL {X  -162.820, Y  +503.236, Z    +0.000, E1   +58.858, E3 +205980.027}
ENDSPLINE

SPLINE
SPL {X  -162.820, Y  +486.621, Z    +0.000, E1   +59.661, E3 +205995.199}
SPL {X  -162.820, Y  +472.771, Z    +0.000, E1   +60.369, E3 +206006.945}
SPL {X  -162.820, Y  +460.138, Z    +0.000, E1   +61.014, E3 +206017.264}
SPL {X  -162.820, Y  +442.137, Z    +0.000, E1   +61.946, E3 +206031.161}
SPL {X  -162.820, Y  +425.982, Z    +0.000, E1   +62.713, E3 +206043.187}
SPL {X  -162.820, Y  +413.005, Z    +0.000, E1   +63.234, E3 +206053.202}
SPL {X  -162.820, Y  +396.727, Z    +0.000, E1   +63.972, E3 +206064.553}
SPL {X  -162.820, Y  +382.966, Z    +0.000, E1   +64.511, E3 +206074.275}
SPL {X  -161.867, Y  +362.911, Z    +0.000, E1   +65.480, E3 +206086.349}
SPL {X  -159.475, Y  +347.667, Z    +0.000, E1   +65.889, E3 +206097.268}
SPL {X  -157.043, Y  +337.513, Z    +0.000, E1   +65.541, E3 +206109.346}
SPL {X  -153.776, Y  +326.991, Z    +0.000, E1   +65.023, E3 +206122.586}
SPL {X  -150.991, Y  +319.573, Z    +0.000, E1   +64.614, E3 +206132.040}
SPL {X  -147.832, Y  +312.265, Z    +0.000, E1   +64.201, E3 +206141.446}
SPL {X  -145.264, Y  +306.955, Z    +0.000, E1   +63.555, E3 +206150.052}
SPL {X  -142.454, Y  +301.650, Z    +0.000, E1   +63.360, E3 +206156.056}
SPL {X  -139.696, Y  +296.861, Z    +0.000, E1   +62.910, E3 +206162.823}
SPL {X  -137.330, Y  +293.030, Z    +0.000, E1   +62.290, E3 +206169.448}
SPL {X  -133.474, Y  +287.253, Z    +0.000, E1   +62.192, E3 +206175.187}
SPL {X  -124.928, Y  +276.081, Z    +0.000, E1   +64.269, E3 +206175.894}
SPL {X   -90.696, Y  +245.280, Z    +0.000, E1   +54.124, E3 +206296.612}
ENDSPLINE

SPLINE
SPL {X  -134.058, Y  +288.094, Z    +0.000, E1   +46.503, E3 +206424.126}
SPL {X  -153.979, Y  +327.577, Z    +0.000, E1   +33.452, E3 +206435.666}
SPL {X  -160.130, Y  +351.024, Z    +0.000, E1   +21.715, E3 +206440.096}
SPL {X  -162.127, Y  +365.491, Z    +0.000, E1   +12.692, E3 +206440.020}
SPL {X  -162.801, Y  +378.004, Z    +0.000, E1    +3.811, E3 +206440.436}
SPL {X  -162.820, Y  +382.501, Z    +0.000, E1    +0.028, E3 +206439.854}
SPL {X  -162.820, Y  +385.123, Z    +0.000, E1    -3.284, E3 +206439.532}
SPL {X  -162.820, Y  +390.608, Z    +0.000, E1   -12.198, E3 +206439.445}
SPL {X  -162.820, Y  +396.028, Z    +0.000, E1   -22.022, E3 +206439.313}
SPL {X  -162.820, Y  +402.037, Z    +0.000, E1   -32.247, E3 +206439.251}
SPL {X  -162.820, Y  +411.189, Z    +0.000, E1   -44.140, E3 +206440.581}
SPL {X  -162.820, Y  +422.160, Z    +0.000, E1   -56.042, E3 +206439.052}
SPL {X  -162.820, Y  +475.891, Z    +0.000, E1   -67.666, E3 +206459.371}
SPL {X  -162.820, Y  +573.811, Z    +0.000, E1   -65.269, E3 +206543.969}
SPL {X  -162.820, Y  +580.233, Z    +0.000, E1   -64.427, E3 +206556.676}
SPL {X  -162.820, Y  +590.756, Z    +0.000, E1   -64.410, E3 +206567.244}
SPL {X  -162.820, Y  +600.605, Z    +0.000, E1   -64.446, E3 +206576.817}
SPL {X  -162.820, Y  +611.699, Z    +0.000, E1   -64.369, E3 +206588.496}
SPL {X  -162.820, Y  +622.825, Z    +0.000, E1   -64.446, E3 +206598.941}
SPL {X  -162.820, Y  +635.776, Z    +0.000, E1   -64.495, E3 +206611.631}
SPL {X  -162.820, Y  +648.933, Z    +0.000, E1   -64.417, E3 +206625.178}
SPL {X  -162.820, Y  +658.800, Z    +0.000, E1   -64.418, E3 +206634.992}
SPL {X  -162.820, Y  +670.777, Z    +0.000, E1   -64.432, E3 +206646.905}
SPL {X  -162.296, Y  +686.556, Z    +0.000, E1   -64.388, E3 +206663.108}
SPL {X  -160.469, Y  +701.070, Z    +0.000, E1   -64.058, E3 +206680.011}
SPL {X  -157.811, Y  +713.575, Z    +0.000, E1   -63.758, E3 +206694.590}
SPL {X  -154.601, Y  +724.576, Z    +0.000, E1   -63.303, E3 +206708.712}
SPL {X  -151.802, Y  +732.376, Z    +0.000, E1   -62.761, E3 +206719.839}
SPL {X  -149.758, Y  +737.398, Z    +0.000, E1   -62.434, E3 +206726.860}
SPL {X  -146.903, Y  +743.713, Z    +0.000, E1   -62.188, E3 +206734.633}
SPL {X  -143.515, Y  +750.401, Z    +0.000, E1   -61.484, E3 +206745.317}
SPL {X  -138.985, Y  +758.314, Z    +0.000, E1   -60.770, E3 +206756.876}
SPL {X  -133.449, Y  +766.783, Z    +0.000, E1   -60.899, E3 +206764.496}
SPL {X   -94.739, Y  +805.919, Z    +0.000, E1   -54.063, E3 +206872.553}
ENDSPLINE

SPLINE
SPL {X  -130.051, Y  +771.465, Z    +0.000, E1   -46.832, E3 +206994.337}
SPL {X  -154.243, Y  +725.647, Z    +0.000, E1   -32.659, E3 +207015.899}
SPL {X  -160.324, Y  +701.901, Z    +0.000, E1   -20.534, E3 +207016.722}
SPL {X  -161.938, Y  +690.423, Z    +0.000, E1   -13.625, E3 +207018.112}
SPL {X  -162.638, Y  +681.194, Z    +0.000, E1    -7.430, E3 +207017.933}
SPL {X  -162.820, Y  +672.793, Z    +0.000, E1    -1.263, E3 +207017.991}
SPL {X  -162.820, Y  +670.674, Z    +0.000, E1    +0.808, E3 +207017.521}
SPL {X  -162.820, Y  +666.307, Z    +0.000, E1    +6.851, E3 +207017.304}
SPL {X  -162.820, Y  +660.761, Z    +0.000, E1   +16.102, E3 +207017.446}
SPL {X  -162.820, Y  +655.024, Z    +0.000, E1   +25.730, E3 +207017.608}
SPL {X  -162.820, Y  +646.498, Z    +0.000, E1   +39.738, E3 +207016.129}
SPL {X  -162.820, Y  +637.711, Z    +0.000, E1   +46.793, E3 +207020.621}
SPL {X  -162.820, Y  +598.602, Z    +0.000, E1   +67.541, E3 +207023.172}
SPL {X  -162.820, Y  +578.435, Z    +0.000, E1   +65.472, E3 +207041.272}
SPL {X  -162.820, Y  +480.401, Z    +0.000, E1   +65.660, E3 +207117.201}
ENDSPLINE

SPLINE
SPL {X  -162.820, Y  +490.253, Z    +0.000, E1   +62.754, E3 +207128.964}
SPL {X  -162.820, Y  +503.236, Z    +0.000, E1   +58.858, E3 +207141.317}
ENDSPLINE

SPLINE
SPL {X  -162.820, Y  +486.621, Z    +0.000, E1   +59.661, E3 +207156.490}
SPL {X  -162.820, Y  +472.771, Z    +0.000, E1   +60.369, E3 +207168.235}
SPL {X  -162.820, Y  +460.138, Z    +0.000, E1   +61.014, E3 +207178.555}
SPL {X  -162.820, Y  +448.741, Z    +0.000, E1   +61.510, E3 +207188.069}
SPL {X  -162.820, Y  +430.985, Z    +0.000, E1   +62.533, E3 +207200.502}
SPL {X  -162.820, Y  +413.005, Z    +0.000, E1   +63.234, E3 +207214.492}
SPL {X  -162.820, Y  +396.727, Z    +0.000, E1   +63.972, E3 +207225.844}
SPL {X  -162.756, Y  +375.937, Z    +0.000, E1   +64.914, E3 +207239.453}
SPL {X  -161.353, Y  +358.691, Z    +0.000, E1   +65.588, E3 +207250.677}
SPL {X  -159.475, Y  +347.667, Z    +0.000, E1   +65.889, E3 +207258.558}
SPL {X  -157.043, Y  +337.513, Z    +0.000, E1   +65.541, E3 +207270.636}
SPL {X  -154.736, Y  +329.832, Z    +0.000, E1   +65.034, E3 +207281.082}
SPL {X  -151.631, Y  +321.184, Z    +0.000, E1   +64.776, E3 +207290.927}
SPL {X  -147.832, Y  +312.265, Z    +0.000, E1   +64.201, E3 +207302.736}
SPL {X  -145.264, Y  +306.955, Z    +0.000, E1   +63.555, E3 +207311.342}
SPL {X  -142.454, Y  +301.650, Z    +0.000, E1   +63.360, E3 +207317.346}
SPL {X  -139.696, Y  +296.861, Z    +0.000, E1   +62.910, E3 +207324.114}
SPL {X  -137.330, Y  +293.030, Z    +0.000, E1   +62.290, E3 +207330.739}
SPL {X  -134.245, Y  +288.366, Z    +0.000, E1   +62.031, E3 +207336.220}
SPL {X  -128.642, Y  +280.693, Z    +0.000, E1   +63.351, E3 +207337.214}
SPL {X   -90.696, Y  +245.280, Z    +0.000, E1   +54.124, E3 +207457.902}
ENDSPLINE

SPLINE
SPL {X  -134.058, Y  +288.094, Z    +0.000, E1   +46.503, E3 +207585.416}
SPL {X  -153.979, Y  +327.577, Z    +0.000, E1   +33.452, E3 +207596.956}
SPL {X  -160.130, Y  +351.024, Z    +0.000, E1   +21.715, E3 +207601.386}
SPL {X  -162.127, Y  +365.491, Z    +0.000, E1   +12.692, E3 +207601.310}
SPL {X  -162.745, Y  +375.564, Z    +0.000, E1    +5.577, E3 +207601.920}
SPL {X  -162.820, Y  +382.222, Z    +0.000, E1    +0.380, E3 +207601.193}
SPL {X  -162.820, Y  +384.010, Z    +0.000, E1    -1.878, E3 +207600.856}
SPL {X  -162.820, Y  +387.631, Z    +0.000, E1    -7.169, E3 +207600.809}
SPL {X  -162.820, Y  +394.064, Z    +0.000, E1   -18.298, E3 +207600.619}
SPL {X  -162.820, Y  +402.037, Z    +0.000, E1   -32.247, E3 +207600.541}
SPL {X  -162.820, Y  +411.189, Z    +0.000, E1   -44.140, E3 +207601.871}
SPL {X  -162.820, Y  +422.160, Z    +0.000, E1   -56.042, E3 +207600.343}
SPL {X  -162.820, Y  +475.891, Z    +0.000, E1   -67.666, E3 +207620.661}
SPL {X  -162.820, Y  +573.811, Z    +0.000, E1   -65.269, E3 +207705.260}
SPL {X  -162.820, Y  +580.233, Z    +0.000, E1   -64.427, E3 +207717.966}
SPL {X  -162.820, Y  +590.756, Z    +0.000, E1   -64.410, E3 +207728.534}
SPL {X  -162.820, Y  +600.605, Z    +0.000, E1   -64.446, E3 +207738.107}
SPL {X  -162.820, Y  +611.699, Z    +0.000, E1   -64.369, E3 +207749.787}
SPL {X  -162.820, Y  +622.825, Z    +0.000, E1   -64.446, E3 +207760.231}
SPL {X  -162.820, Y  +635.776, Z    +0.000, E1   -64.495, E3 +207772.921}
SPL {X  -162.820, Y  +648.933, Z    +0.000, E1   -64.417, E3 +207786.468}
SPL {X  -162.820, Y  +658.800, Z    +0.000, E1   -64.418, E3 +207796.282}
SPL {X  -162.820, Y  +670.777, Z    +0.000, E1   -64.432, E3 +207808.195}
SPL {X  -162.296, Y  +686.556, Z    +0.000, E1   -64.388, E3 +207824.399}
SPL {X  -160.469, Y  +701.070, Z    +0.000, E1   -64.058, E3 +207841.302}
SPL {X  -157.811, Y  +713.575, Z    +0.000, E1   -63.758, E3 +207855.880}
SPL {X  -155.696, Y  +721.135, Z    +0.000, E1   -63.387, E3 +207865.814}
SPL {X  -153.915, Y  +726.609, Z    +0.000, E1   -63.196, E3 +207872.588}
SPL {X  -151.802, Y  +732.376, Z    +0.000, E1   -62.761, E3 +207881.130}
SPL {X  -149.758, Y  +737.398, Z    +0.000, E1   -62.434, E3 +207888.150}
SPL {X  -146.903, Y  +743.713, Z    +0.000, E1   -62.188, E3 +207895.923}
SPL {X  -144.901, Y  +747.758, Z    +0.000, E1   -61.566, E3 +207903.386}
SPL {X  -141.375, Y  +754.268, Z    +0.000, E1   -61.208, E3 +207911.940}
SPL {X  -137.124, Y  +761.291, Z    +0.000, E1   -60.398, E3 +207922.851}
SPL {X  -130.896, Y  +770.333, Z    +0.000, E1   -61.755, E3 +207925.526}
SPL {X   -94.739, Y  +805.919, Z    +0.000, E1   -54.063, E3 +208033.843}
ENDSPLINE

SPLINE
SPL {X  -130.051, Y  +771.465, Z    +0.000, E1   -46.832, E3 +208155.627}
SPL {X  -150.288, Y  +736.141, Z    +0.000, E1   -36.889, E3 +208175.483}
SPL {X  -159.122, Y  +708.003, Z    +0.000, E1   -24.018, E3 +208178.191}
SPL {X  -161.938, Y  +690.423, Z    +0.000, E1   -13.625, E3 +208179.402}
SPL {X  -162.746, Y  +678.392, Z    +0.000, E1    -5.513, E3 +208179.475}
SPL {X  -162.820, Y  +671.700, Z    +0.000, E1    -0.272, E3 +208179.041}
SPL {X  -162.820, Y  +668.888, Z    +0.000, E1    +3.063, E3 +208178.738}
SPL {X  -162.820, Y  +664.763, Z    +0.000, E1    +9.526, E3 +208178.397}
SPL {X  -162.820, Y  +660.761, Z    +0.000, E1   +16.102, E3 +208178.737}
SPL {X  -162.820, Y  +655.024, Z    +0.000, E1   +25.730, E3 +208178.898}
SPL {X  -162.820, Y  +646.498, Z    +0.000, E1   +39.738, E3 +208177.419}
SPL {X  -162.820, Y  +637.711, Z    +0.000, E1   +46.793, E3 +208181.912}
SPL {X  -162.820, Y  +613.264, Z    +0.000, E1   +68.325, E3 +208174.110}
SPL {X  -162.820, Y  +583.199, Z    +0.000, E1   +66.160, E3 +208197.600}
SPL {X  -162.820, Y  +480.401, Z    +0.000, E1   +65.660, E3 +208278.491}
ENDSPLINE

SPLINE
SPL {X  -162.820, Y  +490.253, Z    +0.000, E1   +62.754, E3 +208290.254}
SPL {X  -162.820, Y  +503.236, Z    +0.000, E1   +58.858, E3 +208302.607}
ENDSPLINE

SPLINE
SPL {X  -162.820, Y  +486.621, Z    +0.000, E1   +59.661, E3 +208317.780}
SPL {X  -162.820, Y  +472.771, Z    +0.000, E1   +60.369, E3 +208329.525}
SPL {X  -162.820, Y  +460.138, Z    +0.000, E1   +61.014, E3 +208339.845}
SPL {X  -162.820, Y  +448.741, Z    +0.000, E1   +61.510, E3 +208349.360}
SPL {X  -162.820, Y  +430.985, Z    +0.000, E1   +62.533, E3 +208361.793}
SPL {X  -162.820, Y  +413.005, Z    +0.000, E1   +63.234, E3 +208375.783}
SPL {X  -162.820, Y  +396.727, Z    +0.000, E1   +63.972, E3 +208387.134}
SPL {X  -162.756, Y  +375.937, Z    +0.000, E1   +64.914, E3 +208400.743}
SPL {X  -161.353, Y  +358.691, Z    +0.000, E1   +65.588, E3 +208411.968}
SPL {X  -159.475, Y  +347.667, Z    +0.000, E1   +65.889, E3 +208419.848}
SPL {X  -157.043, Y  +337.513, Z    +0.000, E1   +65.541, E3 +208431.926}
SPL {X  -153.776, Y  +326.991, Z    +0.000, E1   +65.023, E3 +208445.167}
SPL {X  -149.992, Y  +317.154, Z    +0.000, E1   +64.515, E3 +208457.631}
SPL {X  -146.026, Y  +308.480, Z    +0.000, E1   +63.813, E3 +208469.873}
SPL {X  -142.454, Y  +301.650, Z    +0.000, E1   +63.360, E3 +208478.636}
SPL {X  -139.696, Y  +296.861, Z    +0.000, E1   +62.910, E3 +208485.404}
SPL {X  -137.330, Y  +293.030, Z    +0.000, E1   +62.290, E3 +208492.029}
SPL {X  -134.245, Y  +288.366, Z    +0.000, E1   +62.031, E3 +208497.510}
SPL {X  -128.642, Y  +280.693, Z    +0.000, E1   +63.351, E3 +208498.504}
SPL {X   -90.696, Y  +245.280, Z    +0.000, E1   +54.124, E3 +208619.193}
ENDSPLINE

SPLINE
SPL {X  -134.058, Y  +288.094, Z    +0.000, E1   +46.503, E3 +208746.706}
SPL {X  -148.633, Y  +314.028, Z    +0.000, E1   +38.752, E3 +208755.595}
SPL {X  -156.325, Y  +334.971, Z    +0.000, E1   +30.037, E3 +208759.363}
SPL {X  -160.130, Y  +351.024, Z    +0.000, E1   +21.715, E3 +208762.677}
SPL {X  -162.127, Y  +365.491, Z    +0.000, E1   +12.692, E3 +208762.601}
SPL {X  -162.801, Y  +378.004, Z    +0.000, E1    +3.811, E3 +208763.017}
SPL {X  -162.820, Y  +382.997, Z    +0.000, E1    -0.389, E3 +208762.340}
SPL {X  -162.820, Y  +386.358, Z    +0.000, E1    -5.320, E3 +208762.075}
SPL {X  -162.820, Y  +390.608, Z    +0.000, E1   -12.198, E3 +208762.026}
SPL {X  -162.820, Y  +396.028, Z    +0.000, E1   -22.022, E3 +208761.894}
SPL {X  -162.820, Y  +402.037, Z    +0.000, E1   -32.247, E3 +208761.832}
SPL {X  -162.820, Y  +411.189, Z    +0.000, E1   -44.140, E3 +208763.161}
SPL {X  -162.820, Y  +422.160, Z    +0.000, E1   -56.042, E3 +208761.633}
SPL {X  -162.820, Y  +475.891, Z    +0.000, E1   -67.666, E3 +208781.952}
SPL {X  -162.820, Y  +576.352, Z    +0.000, E1   -67.140, E3 +208854.326}
ENDSPLINE

SPLINE
SPL {X  -162.820, Y  +573.336, Z    +0.000, E1   -64.995, E3 +208868.078}
ENDSPLINE

SPLINE
SPL {X  -162.820, Y  +580.233, Z    +0.000, E1   -64.427, E3 +208879.257}
SPL {X  -162.820, Y  +590.756, Z    +0.000, E1   -64.410, E3 +208889.824}
SPL {X  -162.820, Y  +600.605, Z    +0.000, E1   -64.446, E3 +208899.397}
SPL {X  -162.820, Y  +611.699, Z    +0.000, E1   -64.369, E3 +208911.077}
SPL {X  -162.820, Y  +625.950, Z    +0.000, E1   -64.427, E3 +208924.917}
SPL {X  -162.820, Y  +639.401, Z    +0.000, E1   -64.540, E3 +208937.340}
SPL {X  -162.820, Y  +648.933, Z    +0.000, E1   -64.417, E3 +208947.758}
SPL {X  -162.820, Y  +658.800, Z    +0.000, E1   -64.418, E3 +208957.572}
SPL {X  -162.820, Y  +670.777, Z    +0.000, E1   -64.432, E3 +208969.486}
SPL {X  -162.296, Y  +686.556, Z    +0.000, E1   -64.388, E3 +208985.689}
SPL {X  -161.171, Y  +696.611, Z    +0.000, E1   -64.029, E3 +208998.154}
SPL {X  -159.311, Y  +707.123, Z    +0.000, E1   -64.022, E3 +209008.848}
SPL {X  -156.625, Y  +717.984, Z    +0.000, E1   -63.524, E3 +209023.203}
SPL {X  -153.915, Y  +726.609, Z    +0.000, E1   -63.196, E3 +209033.879}
SPL {X  -151.802, Y  +732.376, Z    +0.000, E1   -62.761, E3 +209042.420}
SPL {X  -149.758, Y  +737.398, Z    +0.000, E1   -62.434, E3 +209049.441}
SPL {X  -146.903, Y  +743.713, Z    +0.000, E1   -62.188, E3 +209057.213}
SPL {X  -143.515, Y  +750.401, Z    +0.000, E1   -61.484, E3 +209067.897}
SPL {X  -140.303, Y  +756.116, Z    +0.000, E1   -60.974, E3 +209076.095}
SPL {X  -137.124, Y  +761.291, Z    +0.000, E1   -60.398, E3 +209084.142}
SPL {X  -130.896, Y  +770.333, Z    +0.000, E1   -61.755, E3 +209086.816}
SPL {X   -94.739, Y  +805.919, Z    +0.000, E1   -54.063, E3 +209195.133}
ENDSPLINE

SPLINE
SPL {X  -130.051, Y  +771.465, Z    +0.000, E1   -46.832, E3 +209316.917}
SPL {X  -154.243, Y  +725.647, Z    +0.000, E1   -32.659, E3 +209338.479}
SPL {X  -161.394, Y  +695.005, Z    +0.000, E1   -16.571, E3 +209340.184}
SPL {X  -162.746, Y  +678.392, Z    +0.000, E1    -5.513, E3 +209340.765}
SPL {X  -162.820, Y  +671.700, Z    +0.000, E1    -0.272, E3 +209340.331}
SPL {X  -162.820, Y  +668.888, Z    +0.000, E1    +3.063, E3 +209340.028}
SPL {X  -162.820, Y  +664.763, Z    +0.000, E1    +9.526, E3 +209339.688}
SPL {X  -162.820, Y  +660.761, Z    +0.000, E1   +16.102, E3 +209340.027}
SPL {X  -162.820, Y  +655.024, Z    +0.000, E1   +25.730, E3 +209340.188}
SPL {X  -162.820, Y  +646.498, Z    +0.000, E1   +39.738, E3 +209338.709}
SPL {X  -162.820, Y  +637.711, Z    +0.000, E1   +46.793, E3 +209343.202}
SPL {X  -162.820, Y  +598.602, Z    +0.000, E1   +67.541, E3 +209345.753}
SPL {X  -162.820, Y  +578.435, Z    +0.000, E1   +65.472, E3 +209363.853}
SPL {X  -162.820, Y  +475.450, Z    +0.000, E1   +67.130, E3 +209432.790}
ENDSPLINE

SPLINE
SPL {X  -162.820, Y  +483.223, Z    +0.000, E1   +64.312, E3 +209447.230}
SPL {X  -162.820, Y  +502.830, Z    +0.000, E1   +59.229, E3 +209462.151}
ENDSPLINE

SPLINE
SPL {X  -162.820, Y  +486.621, Z    +0.000, E1   +59.661, E3 +209479.070}
SPL {X  -162.820, Y  +472.771, Z    +0.000, E1   +60.369, E3 +209490.816}
SPL {X  -162.820, Y  +460.138, Z    +0.000, E1   +61.014, E3 +209501.135}
SPL {X  -162.820, Y  +448.741, Z    +0.000, E1   +61.510, E3 +209510.650}
SPL {X  -162.820, Y  +430.985, Z    +0.000, E1   +62.533, E3 +209523.083}
SPL {X  -162.820, Y  +413.005, Z    +0.000, E1   +63.234, E3 +209537.073}
SPL {X  -162.820, Y  +396.727, Z    +0.000, E1   +63.972, E3 +209548.424}
SPL {X  -162.820, Y  +382.966, Z    +0.000, E1   +64.511, E3 +209558.146}
SPL {X  -161.867, Y  +362.911, Z    +0.000, E1   +65.480, E3 +209570.220}
SPL {X  -159.475, Y  +347.667, Z    +0.000, E1   +65.889, E3 +209581.139}
SPL {X  -157.043, Y  +337.513, Z    +0.000, E1   +65.541, E3 +209593.217}
SPL {X  -153.776, Y  +326.991, Z    +0.000, E1   +65.023, E3 +209606.457}
SPL {X  -150.991, Y  +319.573, Z    +0.000, E1   +64.614, E3 +209615.911}
SPL {X  -147.832, Y  +312.265, Z    +0.000, E1   +64.201, E3 +209625.317}
SPL {X  -145.264, Y  +306.955, Z    +0.000, E1   +63.555, E3 +209633.923}
SPL {X  -142.454, Y  +301.650, Z    +0.000, E1   +63.360, E3 +209639.927}
SPL {X  -139.696, Y  +296.861, Z    +0.000, E1   +62.910, E3 +209646.694}
SPL {X  -137.330, Y  +293.030, Z    +0.000, E1   +62.290, E3 +209653.319}
SPL {X  -133.474, Y  +287.253, Z    +0.000, E1   +62.192, E3 +209659.058}
SPL {X  -124.928, Y  +276.081, Z    +0.000, E1   +64.269, E3 +209659.765}
SPL {X   -90.696, Y  +245.280, Z    +0.000, E1   +54.124, E3 +209780.483}
ENDSPLINE

SPLINE
SPL {X  -134.058, Y  +288.094, Z    +0.000, E1   +46.503, E3 +209907.997}
SPL {X  -153.979, Y  +327.577, Z    +0.000, E1   +33.452, E3 +209919.537}
SPL {X  -160.130, Y  +351.024, Z    +0.000, E1   +21.715, E3 +209923.967}
SPL {X  -162.127, Y  +365.491, Z    +0.000, E1   +12.692, E3 +209923.891}
SPL {X  -162.801, Y  +378.004, Z    +0.000, E1    +3.811, E3 +209924.307}
SPL {X  -162.820, Y  +382.997, Z    +0.000, E1    -0.389, E3 +209923.630}
SPL {X  -162.820, Y  +386.358, Z    +0.000, E1    -5.320, E3 +209923.365}
SPL {X  -162.820, Y  +390.608, Z    +0.000, E1   -12.198, E3 +209923.316}
SPL {X  -162.820, Y  +396.028, Z    +0.000, E1   -22.022, E3 +209923.184}
SPL {X  -162.820, Y  +402.037, Z    +0.000, E1   -32.247, E3 +209923.122}
SPL {X  -162.820, Y  +414.067, Z    +0.000, E1   -47.235, E3 +209924.548}
SPL {X  -162.820, Y  +424.566, Z    +0.000, E1   -59.255, E3 +209921.213}
SPL {X  -162.820, Y  +460.664, Z    +0.000, E1   -69.605, E3 +209929.509}
SPL {X  -162.820, Y  +481.040, Z    +0.000, E1   -67.047, E3 +209948.098}
SPL {X  -162.820, Y  +576.352, Z    +0.000, E1   -67.140, E3 +210015.617}
ENDSPLINE

SPLINE
SPL {X  -162.820, Y  +573.336, Z    +0.000, E1   -64.995, E3 +210029.369}
ENDSPLINE

SPLINE
SPL {X  -162.820, Y  +580.233, Z    +0.000, E1   -64.427, E3 +210040.547}
SPL {X  -162.820, Y  +590.756, Z    +0.000, E1   -64.410, E3 +210051.115}
SPL {X  -162.820, Y  +600.605, Z    +0.000, E1   -64.446, E3 +210060.688}
SPL {X  -162.820, Y  +611.699, Z    +0.000, E1   -64.369, E3 +210072.367}
SPL {X  -162.820, Y  +625.950, Z    +0.000, E1   -64.427, E3 +210086.208}
SPL {X  -162.820, Y  +639.401, Z    +0.000, E1   -64.540, E3 +210098.630}
SPL {X  -162.820, Y  +648.933, Z    +0.000, E1   -64.417, E3 +210109.049}
SPL {X  -162.820, Y  +658.800, Z    +0.000, E1   -64.418, E3 +210118.863}
SPL {X  -162.820, Y  +670.777, Z    +0.000, E1   -64.432, E3 +210130.776}
SPL {X  -162.296, Y  +686.556, Z    +0.000, E1   -64.388, E3 +210146.979}
SPL {X  -160.469, Y  +701.070, Z    +0.000, E1   -64.058, E3 +210163.882}
SPL {X  -157.811, Y  +713.575, Z    +0.000, E1   -63.758, E3 +210178.461}
SPL {X  -154.601, Y  +724.576, Z    +0.000, E1   -63.303, E3 +210192.583}
SPL {X  -151.802, Y  +732.376, Z    +0.000, E1   -62.761, E3 +210203.710}
SPL {X  -149.758, Y  +737.398, Z    +0.000, E1   -62.434, E3 +210210.731}
SPL {X  -146.903, Y  +743.713, Z    +0.000, E1   -62.188, E3 +210218.504}
SPL {X  -143.515, Y  +750.401, Z    +0.000, E1   -61.484, E3 +210229.188}
SPL {X  -138.985, Y  +758.314, Z    +0.000, E1   -60.770, E3 +210240.747}
SPL {X  -133.449, Y  +766.783, Z    +0.000, E1   -60.899, E3 +210248.367}
SPL {X   -94.739, Y  +805.919, Z    +0.000, E1   -54.063, E3 +210356.424}
ENDSPLINE

SPLINE
SPL {X  -130.051, Y  +771.465, Z    +0.000, E1   -46.832, E3 +210478.207}
SPL {X  -150.288, Y  +736.141, Z    +0.000, E1   -36.889, E3 +210498.063}
SPL {X  -159.122, Y  +708.003, Z    +0.000, E1   -24.018, E3 +210500.772}
SPL {X  -161.938, Y  +690.423, Z    +0.000, E1   -13.625, E3 +210501.983}
SPL {X  -162.638, Y  +681.194, Z    +0.000, E1    -7.430, E3 +210501.804}
SPL {X  -162.805, Y  +675.686, Z    +0.000, E1    -3.400, E3 +210502.280}
SPL {X  -162.820, Y  +671.700, Z    +0.000, E1    -0.272, E3 +210501.621}
SPL {X  -162.820, Y  +668.888, Z    +0.000, E1    +3.063, E3 +210501.319}
SPL {X  -162.820, Y  +664.763, Z    +0.000, E1    +9.526, E3 +210500.978}
SPL {X  -162.820, Y  +659.878, Z    +0.000, E1   +17.497, E3 +210501.383}
SPL {X  -162.820, Y  +650.308, Z    +0.000, E1   +33.487, E3 +210500.796}
SPL {X  -162.820, Y  +637.711, Z    +0.000, E1   +46.793, E3 +210504.492}
SPL {X  -162.820, Y  +598.602, Z    +0.000, E1   +67.541, E3 +210507.043}
SPL {X  -162.820, Y  +578.435, Z    +0.000, E1   +65.472, E3 +210525.143}
SPL {X  -162.820, Y  +475.450, Z    +0.000, E1   +67.130, E3 +210594.081}
ENDSPLINE

SPLINE
SPL {X  -162.820, Y  +483.223, Z    +0.000, E1   +64.312, E3 +210608.520}
SPL {X  -162.820, Y  +502.830, Z    +0.000, E1   +59.229, E3 +210623.441}
ENDSPLINE

SPLINE
SPL {X  -162.820, Y  +486.621, Z    +0.000, E1   +59.661, E3 +210640.360}
SPL {X  -162.820, Y  +472.771, Z    +0.000, E1   +60.369, E3 +210652.106}
SPL {X  -162.820, Y  +460.138, Z    +0.000, E1   +61.014, E3 +210662.425}
SPL {X  -162.820, Y  +448.741, Z    +0.000, E1   +61.510, E3 +210671.940}
SPL {X  -162.820, Y  +430.985, Z    +0.000, E1   +62.533, E3 +210684.373}
SPL {X  -162.820, Y  +413.005, Z    +0.000, E1   +63.234, E3 +210698.363}
SPL {X  -162.820, Y  +396.727, Z    +0.000, E1   +63.972, E3 +210709.715}
SPL {X  -162.756, Y  +375.937, Z    +0.000, E1   +64.914, E3 +210723.324}
SPL {X  -161.353, Y  +358.691, Z    +0.000, E1   +65.588, E3 +210734.548}
SPL {X  -159.475, Y  +347.667, Z    +0.000, E1   +65.889, E3 +210742.429}
SPL {X  -157.043, Y  +337.513, Z    +0.000, E1   +65.541, E3 +210754.507}
SPL {X  -153.776, Y  +326.991, Z    +0.000, E1   +65.023, E3 +210767.747}
SPL {X  -149.992, Y  +317.154, Z    +0.000, E1   +64.515, E3 +210780.211}
SPL {X  -146.026, Y  +308.480, Z    +0.000, E1   +63.813, E3 +210792.453}
SPL {X  -142.454, Y  +301.650, Z    +0.000, E1   +63.360, E3 +210801.217}
SPL {X  -139.696, Y  +296.861, Z    +0.000, E1   +62.910, E3 +210807.985}
SPL {X  -137.330, Y  +293.030, Z    +0.000, E1   +62.290, E3 +210814.610}
SPL {X  -134.245, Y  +288.366, Z    +0.000, E1   +62.031, E3 +210820.091}
SPL {X  -128.642, Y  +280.693, Z    +0.000, E1   +63.351, E3 +210821.085}
SPL {X   -90.696, Y  +245.280, Z    +0.000, E1   +54.124, E3 +210941.773}
ENDSPLINE

SPLINE
SPL {X  -134.058, Y  +288.094, Z    +0.000, E1   +46.503, E3 +211069.287}
SPL {X  -153.979, Y  +327.577, Z    +0.000, E1   +33.452, E3 +211080.827}
SPL {X  -160.130, Y  +351.024, Z    +0.000, E1   +21.715, E3 +211085.257}
SPL {X  -162.127, Y  +365.491, Z    +0.000, E1   +12.692, E3 +211085.181}
SPL {X  -162.745, Y  +375.564, Z    +0.000, E1    +5.577, E3 +211085.791}
SPL {X  -162.820, Y  +382.222, Z    +0.000, E1    +0.380, E3 +211085.064}
SPL {X  -162.820, Y  +385.123, Z    +0.000, E1    -3.284, E3 +211084.693}
SPL {X  -162.820, Y  +390.608, Z    +0.000, E1   -12.198, E3 +211084.607}
SPL {X  -162.820, Y  +396.028, Z    +0.000, E1   -22.022, E3 +211084.474}
SPL {X  -162.820, Y  +402.037, Z    +0.000, E1   -32.247, E3 +211084.412}
SPL {X  -162.820, Y  +411.189, Z    +0.000, E1   -44.140, E3 +211085.742}
SPL {X  -162.820, Y  +422.160, Z    +0.000, E1   -56.042, E3 +211084.214}
SPL {X  -162.820, Y  +475.891, Z    +0.000, E1   -67.666, E3 +211104.532}
SPL {X  -162.820, Y  +576.352, Z    +0.000, E1   -67.140, E3 +211176.907}
ENDSPLINE

SPLINE
SPL {X  -162.820, Y  +573.336, Z    +0.000, E1   -64.995, E3 +211190.659}
ENDSPLINE

SPLINE
SPL {X  -162.820, Y  +580.233, Z    +0.000, E1   -64.427, E3 +211201.837}
SPL {X  -162.820, Y  +590.756, Z    +0.000, E1   -64.410, E3 +211212.405}
SPL {X  -162.820, Y  +600.605, Z    +0.000, E1   -64.446, E3 +211221.978}
SPL {X  -162.820, Y  +611.699, Z    +0.000, E1   -64.369, E3 +211233.658}
SPL {X  -162.820, Y  +622.825, Z    +0.000, E1   -64.446, E3 +211244.102}
SPL {X  -162.820, Y  +635.776, Z    +0.000, E1   -64.495, E3 +211256.792}
SPL {X  -162.820, Y  +648.933, Z    +0.000, E1   -64.417, E3 +211270.339}
SPL {X  -162.820, Y  +658.800, Z    +0.000, E1   -64.418, E3 +211280.153}
SPL {X  -162.820, Y  +670.777, Z    +0.000, E1   -64.432, E3 +211292.066}
SPL {X  -162.613, Y  +681.710, Z    +0.000, E1   -64.310, E3 +211303.830}
SPL {X  -161.587, Y  +693.503, Z    +0.000, E1   -64.259, E3 +211316.184}
SPL {X  -159.883, Y  +704.285, Z    +0.000, E1   -64.016, E3 +211328.525}
SPL {X  -157.811, Y  +713.575, Z    +0.000, E1   -63.758, E3 +211339.751}
SPL {X  -154.601, Y  +724.576, Z    +0.000, E1   -63.303, E3 +211353.874}
SPL {X  -151.802, Y  +732.376, Z    +0.000, E1   -62.761, E3 +211365.001}
SPL {X  -149.758, Y  +737.398, Z    +0.000, E1   -62.434, E3 +211372.021}
SPL {X  -146.903, Y  +743.713, Z    +0.000, E1   -62.188, E3 +211379.794}
SPL {X  -144.901, Y  +747.758, Z    +0.000, E1   -61.566, E3 +211387.257}
SPL {X  -141.375, Y  +754.268, Z    +0.000, E1   -61.208, E3 +211395.811}
SPL {X  -137.124, Y  +761.291, Z    +0.000, E1   -60.398, E3 +211406.722}
SPL {X  -130.896, Y  +770.333, Z    +0.000, E1   -61.755, E3 +211409.397}
SPL {X   -94.739, Y  +805.919, Z    +0.000, E1   -54.063, E3 +211517.714}
ENDSPLINE

SPLINE
SPL {X  -120.571, Y  +782.921, Z    +0.000, E1   -48.746, E3 +211625.010}
SPL {X  -145.902, Y  +745.770, Z    +0.000, E1   -40.275, E3 +211656.158}
SPL {X  -156.935, Y  +716.881, Z    +0.000, E1   -28.554, E3 +211662.146}
SPL {X  -161.394, Y  +695.005, Z    +0.000, E1   -16.571, E3 +211662.765}
SPL {X  -162.746, Y  +678.392, Z    +0.000, E1    -5.513, E3 +211663.346}
SPL {X  -162.820, Y  +671.700, Z    +0.000, E1    -0.272, E3 +211662.911}
SPL {X  -162.820, Y  +669.993, Z    +0.000, E1    +1.755, E3 +211662.578}
SPL {X  -162.820, Y  +666.307, Z    +0.000, E1    +6.851, E3 +211662.465}
SPL {X  -162.820, Y  +659.878, Z    +0.000, E1   +17.497, E3 +211662.673}
SPL {X  -162.820, Y  +650.308, Z    +0.000, E1   +33.487, E3 +211662.087}
SPL {X  -162.820, Y  +637.711, Z    +0.000, E1   +46.793, E3 +211665.782}
SPL {X  -162.820, Y  +613.264, Z    +0.000, E1   +68.325, E3 +211657.981}
SPL {X  -162.820, Y  +583.199, Z    +0.000, E1   +66.160, E3 +211681.471}
SPL {X  -162.820, Y  +480.401, Z    +0.000, E1   +65.660, E3 +211762.362}
ENDSPLINE

SPLINE
SPL {X  -162.820, Y  +490.253, Z    +0.000, E1   +62.754, E3 +211774.125}
SPL {X  -162.820, Y  +503.236, Z    +0.000, E1   +58.858, E3 +211786.478}
ENDSPLINE

SPLINE
SPL {X  -162.820, Y  +486.621, Z    +0.000, E1   +59.661, E3 +211801.651}
SPL {X  -162.820, Y  +472.771, Z    +0.000, E1   +60.369, E3 +211813.396}
SPL {X  -162.820, Y  +460.138, Z    +0.000, E1   +61.014, E3 +211823.716}
SPL {X  -162.820, Y  +442.137, Z    +0.000, E1   +61.946, E3 +211837.613}
SPL {X  -162.820, Y  +425.982, Z    +0.000, E1   +62.713, E3 +211849.639}
SPL {X  -162.820, Y  +413.005, Z    +0.000, E1   +63.234, E3 +211859.654}
SPL {X  -162.820, Y  +396.727, Z    +0.000, E1   +63.972, E3 +211871.005}
SPL {X  -162.820, Y  +382.966, Z    +0.000, E1   +64.511, E3 +211880.727}
SPL {X  -161.867, Y  +362.911, Z    +0.000, E1   +65.480, E3 +211892.801}
SPL {X  -159.475, Y  +347.667, Z    +0.000, E1   +65.889, E3 +211903.719}
SPL {X  -157.043, Y  +337.513, Z    +0.000, E1   +65.541, E3 +211915.797}
SPL {X  -153.776, Y  +326.991, Z    +0.000, E1   +65.023, E3 +211929.038}
SPL {X  -150.991, Y  +319.573, Z    +0.000, E1   +64.614, E3 +211938.492}
SPL {X  -147.832, Y  +312.265, Z    +0.000, E1   +64.201, E3 +211947.898}
SPL {X  -145.264, Y  +306.955, Z    +0.000, E1   +63.555, E3 +211956.504}
SPL {X  -142.454, Y  +301.650, Z    +0.000, E1   +63.360, E3 +211962.507}
SPL {X  -139.696, Y  +296.861, Z    +0.000, E1   +62.910, E3 +211969.275}
SPL {X  -137.330, Y  +293.030, Z    +0.000, E1   +62.290, E3 +211975.900}
SPL {X  -133.474, Y  +287.253, Z    +0.000, E1   +62.192, E3 +211981.639}
SPL {X  -124.928, Y  +276.081, Z    +0.000, E1   +64.269, E3 +211982.346}
SPL {X   -90.696, Y  +245.280, Z    +0.000, E1   +54.124, E3 +212103.064}
ENDSPLINE

SPLINE
SPL {X  -134.058, Y  +288.094, Z    +0.000, E1   +46.503, E3 +212230.577}
SPL {X  -153.979, Y  +327.577, Z    +0.000, E1   +33.452, E3 +212242.117}
SPL {X  -160.130, Y  +351.024, Z    +0.000, E1   +21.715, E3 +212246.548}
SPL {X  -162.127, Y  +365.491, Z    +0.000, E1   +12.692, E3 +212246.471}
SPL {X  -162.801, Y  +378.004, Z    +0.000, E1    +3.811, E3 +212246.887}
SPL {X  -162.820, Y  +382.501, Z    +0.000, E1    +0.028, E3 +212246.306}
SPL {X  -162.820, Y  +385.123, Z    +0.000, E1    -3.284, E3 +212245.983}
SPL {X  -162.820, Y  +390.608, Z    +0.000, E1   -12.198, E3 +212245.897}
SPL {X  -162.820, Y  +396.028, Z    +0.000, E1   -22.022, E3 +212245.765}
SPL {X  -162.820, Y  +402.037, Z    +0.000, E1   -32.247, E3 +212245.703}
SPL {X  -162.820, Y  +411.189, Z    +0.000, E1   -44.140, E3 +212247.032}
SPL {X  -162.820, Y  +422.160, Z    +0.000, E1   -56.042, E3 +212245.504}
SPL {X  -162.820, Y  +475.891, Z    +0.000, E1   -67.666, E3 +212265.823}
SPL {X  -162.820, Y  +573.811, Z    +0.000, E1   -65.269, E3 +212350.421}
SPL {X  -162.820, Y  +580.233, Z    +0.000, E1   -64.427, E3 +212363.128}
SPL {X  -162.820, Y  +590.756, Z    +0.000, E1   -64.410, E3 +212373.695}
SPL {X  -162.820, Y  +600.605, Z    +0.000, E1   -64.446, E3 +212383.268}
SPL {X  -162.820, Y  +611.699, Z    +0.000, E1   -64.369, E3 +212394.948}
SPL {X  -162.820, Y  +622.825, Z    +0.000, E1   -64.446, E3 +212405.393}
SPL {X  -162.820, Y  +635.776, Z    +0.000, E1   -64.495, E3 +212418.082}
SPL {X  -162.820, Y  +648.933, Z    +0.000, E1   -64.417, E3 +212431.629}
SPL {X  -162.820, Y  +658.800, Z    +0.000, E1   -64.418, E3 +212441.443}
SPL {X  -162.820, Y  +670.777, Z    +0.000, E1   -64.432, E3 +212453.357}
SPL {X  -162.296, Y  +686.556, Z    +0.000, E1   -64.388, E3 +212469.560}
SPL {X  -160.469, Y  +701.070, Z    +0.000, E1   -64.058, E3 +212486.463}
SPL {X  -157.811, Y  +713.575, Z    +0.000, E1   -63.758, E3 +212501.042}
SPL {X  -154.601, Y  +724.576, Z    +0.000, E1   -63.303, E3 +212515.164}
SPL {X  -151.802, Y  +732.376, Z    +0.000, E1   -62.761, E3 +212526.291}
SPL {X  -149.758, Y  +737.398, Z    +0.000, E1   -62.434, E3 +212533.311}
SPL {X  -146.903, Y  +743.713, Z    +0.000, E1   -62.188, E3 +212541.084}
SPL {X  -144.901, Y  +747.758, Z    +0.000, E1   -61.566, E3 +212548.547}
SPL {X  -141.375, Y  +754.268, Z    +0.000, E1   -61.208, E3 +212557.101}
SPL {X  -137.988, Y  +759.927, Z    +0.000, E1   -60.537, E3 +212565.900}
SPL {X  -134.516, Y  +765.238, Z    +0.000, E1   -60.629, E3 +212570.703}
SPL {X  -126.113, Y  +776.485, Z    +0.000, E1   -62.672, E3 +212572.263}
SPL {X   -94.739, Y  +805.919, Z    +0.000, E1   -54.063, E3 +212679.004}
ENDSPLINE

SPLINE
SPL {X  -130.051, Y  +771.465, Z    +0.000, E1   -46.832, E3 +212800.788}
SPL {X  -150.288, Y  +736.141, Z    +0.000, E1   -36.889, E3 +212820.644}
SPL {X  -159.122, Y  +708.003, Z    +0.000, E1   -24.018, E3 +212823.353}
SPL {X  -161.938, Y  +690.423, Z    +0.000, E1   -13.625, E3 +212824.564}
SPL {X  -162.746, Y  +678.392, Z    +0.000, E1    -5.513, E3 +212824.636}
SPL {X  -162.820, Y  +672.097, Z    +0.000, E1    -0.584, E3 +212824.341}
SPL {X  -162.820, Y  +670.674, Z    +0.000, E1    +0.808, E3 +212823.973}
SPL {X  -162.820, Y  +666.307, Z    +0.000, E1    +6.851, E3 +212823.755}
SPL {X  -162.820, Y  +660.761, Z    +0.000, E1   +16.102, E3 +212823.898}
SPL {X  -162.820, Y  +655.024, Z    +0.000, E1   +25.730, E3 +212824.059}
SPL {X  -162.820, Y  +646.498, Z    +0.000, E1   +39.738, E3 +212822.580}
SPL {X  -162.820, Y  +637.711, Z    +0.000, E1   +46.793, E3 +212827.073}
SPL {X  -162.820, Y  +613.264, Z    +0.000, E1   +68.325, E3 +212819.271}
SPL {X  -162.820, Y  +583.199, Z    +0.000, E1   +66.160, E3 +212842.761}
SPL {X  -162.820, Y  +480.401, Z    +0.000, E1   +65.660, E3 +212923.653}
ENDSPLINE

SPLINE
SPL {X  -162.820, Y  +490.253, Z    +0.000, E1   +62.754, E3 +212935.415}
SPL {X  -162.820, Y  +505.887, Z    +0.000, E1   +58.743, E3 +212945.106}
ENDSPLINE

SPLINE
SPL {X  -162.820, Y  +492.515, Z    +0.000, E1   +59.352, E3 +212957.790}
SPL {X  -162.820, Y  +476.196, Z    +0.000, E1   +60.204, E3 +212971.823}
SPL {X  -162.820, Y  +460.138, Z    +0.000, E1   +61.014, E3 +212985.006}
SPL {X  -162.820, Y  +442.137, Z    +0.000, E1   +61.946, E3 +212998.903}
SPL {X  -162.820, Y  +425.982, Z    +0.000, E1   +62.713, E3 +213010.929}
SPL {X  -162.820, Y  +413.005, Z    +0.000, E1   +63.234, E3 +213020.944}
SPL {X  -162.820, Y  +396.727, Z    +0.000, E1   +63.972, E3 +213032.295}
SPL {X  -162.820, Y  +382.966, Z    +0.000, E1   +64.511, E3 +213042.017}
SPL {X  -161.867, Y  +362.911, Z    +0.000, E1   +65.480, E3 +213054.091}
ENDSPLINE

SPLINE
SPL {X  -162.496, Y  +370.230, Z    +0.000, E1   +62.662, E3 +213067.266}
ENDSPLINE

SPLINE
SPL {X  -161.953, Y  +363.716, Z    +0.000, E1   +62.355, E3 +213076.531}
SPL {X  -160.528, Y  +353.277, Z    +0.000, E1   +62.144, E3 +213089.527}
SPL {X  -157.973, Y  +341.066, Z    +0.000, E1   +61.800, E3 +213105.126}
SPL {X  -155.627, Y  +332.640, Z    +0.000, E1   +61.354, E3 +213117.040}
SPL {X  -153.198, Y  +325.358, Z    +0.000, E1   +61.117, E3 +213126.470}
SPL {X  -151.022, Y  +319.651, Z    +0.000, E1   +60.776, E3 +213134.643}
SPL {X  -149.105, Y  +315.094, Z    +0.000, E1   +60.301, E3 +213142.396}
SPL {X  -146.196, Y  +308.826, Z    +0.000, E1   +59.961, E3 +213151.103}
SPL {X  -143.704, Y  +303.952, Z    +0.000, E1   +59.374, E3 +213159.460}
SPL {X  -140.940, Y  +298.976, Z    +0.000, E1   +59.075, E3 +213166.385}
SPL {X  -137.763, Y  +293.715, Z    +0.000, E1   +58.761, E3 +213173.492}
SPL {X  -129.725, Y  +282.103, Z    +0.000, E1   +61.069, E3 +213174.995}
SPL {X  -106.695, Y  +257.510, Z    +0.000, E1   +52.408, E3 +213275.717}
SPL {X  -104.122, Y  +255.325, Z    +0.000, E1   +51.312, E3 +213365.775}
ENDSPLINE

SPLINE
SPL {X  -140.007, Y  +297.383, Z    +0.000, E1   +42.766, E3 +213405.100}
SPL {X  -155.551, Y  +332.393, Z    +0.000, E1   +29.794, E3 +213411.021}
SPL {X  -159.755, Y  +349.054, Z    +0.000, E1   +21.610, E3 +213412.894}
SPL {X  -162.078, Y  +364.978, Z    +0.000, E1   +12.369, E3 +213415.631}
SPL {X  -162.752, Y  +375.778, Z    +0.000, E1    +5.236, E3 +213415.340}
SPL {X  -162.820, Y  +381.939, Z    +0.000, E1    +0.593, E3 +213414.967}
SPL {X  -162.820, Y  +383.993, Z    +0.000, E1    -1.497, E3 +213414.540}
SPL {X  -162.820, Y  +388.628, Z    +0.000, E1    -7.678, E3 +213414.443}
SPL {X  -162.820, Y  +394.643, Z    +0.000, E1   -17.317, E3 +213414.243}
SPL {X  -162.820, Y  +401.515, Z    +0.000, E1   -27.960, E3 +213415.063}
SPL {X  -162.820, Y  +412.105, Z    +0.000, E1   -42.847, E3 +213414.055}
SPL {X  -162.820, Y  +422.796, Z    +0.000, E1   -52.392, E3 +213415.276}
SPL {X  -162.820, Y  +474.423, Z    +0.000, E1   -65.078, E3 +213436.326}
SPL {X  -162.820, Y  +578.686, Z    +0.000, E1   -67.085, E3 +213505.491}
ENDSPLINE

SPLINE
SPL {X  -162.820, Y  +565.364, Z    +0.000, E1   -63.589, E3 +213519.491}
ENDSPLINE

SPLINE
SPL {X  -162.820, Y  +574.608, Z    +0.000, E1   -63.370, E3 +213530.750}
SPL {X  -162.820, Y  +584.314, Z    +0.000, E1   -63.342, E3 +213541.042}
SPL {X  -162.820, Y  +593.857, Z    +0.000, E1   -63.382, E3 +213550.744}
SPL {X  -162.820, Y  +602.272, Z    +0.000, E1   -63.279, E3 +213560.272}
SPL {X  -162.820, Y  +613.309, Z    +0.000, E1   -63.489, E3 +213570.271}
SPL {X  -162.820, Y  +627.013, Z    +0.000, E1   -63.389, E3 +213585.492}
SPL {X  -162.820, Y  +642.772, Z    +0.000, E1   -63.348, E3 +213602.150}
SPL {X  -162.820, Y  +658.642, Z    +0.000, E1   -63.324, E3 +213619.066}
SPL {X  -162.819, Y  +673.983, Z    +0.000, E1   -63.398, E3 +213634.393}
SPL {X  -162.617, Y  +681.634, Z    +0.000, E1   -63.169, E3 +213644.015}
SPL {X  -161.618, Y  +693.246, Z    +0.000, E1   -63.233, E3 +213655.873}
SPL {X  -160.212, Y  +702.527, Z    +0.000, E1   -62.898, E3 +213667.818}
SPL {X  -158.647, Y  +710.128, Z    +0.000, E1   -62.776, E3 +213676.640}
SPL {X  -156.957, Y  +716.799, Z    +0.000, E1   -62.460, E3 +213685.759}
SPL {X  -155.130, Y  +722.947, Z    +0.000, E1   -62.207, E3 +213693.871}
SPL {X  -152.287, Y  +731.112, Z    +0.000, E1   -61.798, E3 +213705.146}
SPL {X  -149.420, Y  +738.185, Z    +0.000, E1   -61.282, E3 +213715.555}
SPL {X  -146.960, Y  +743.593, Z    +0.000, E1   -60.951, E3 +213723.099}
SPL {X  -143.277, Y  +750.844, Z    +0.000, E1   -60.348, E3 +213734.105}
SPL {X  -139.430, Y  +757.582, Z    +0.000, E1   -59.554, E3 +213744.980}
SPL {X  -134.550, Y  +765.187, Z    +0.000, E1   -59.954, E3 +213750.931}
SPL {X  -100.103, Y  +801.912, Z    +0.000, E1   -53.794, E3 +213848.981}
ENDSPLINE

SPLINE
SPL {X  -112.938, Y  +790.784, Z    +0.000, E1   -51.983, E3 +213984.503}
SPL {X  -145.058, Y  +747.450, Z    +0.000, E1   -40.634, E3 +213992.613}
SPL {X  -158.857, Y  +709.206, Z    +0.000, E1   -24.633, E3 +214000.582}
SPL {X  -162.312, Y  +686.349, Z    +0.000, E1   -11.031, E3 +214002.151}
SPL {X  -162.811, Y  +675.182, Z    +0.000, E1    -3.078, E3 +214002.226}
SPL {X  -162.820, Y  +671.474, Z    +0.000, E1    -0.022, E3 +214001.696}
SPL {X  -162.820, Y  +668.525, Z    +0.000, E1    +3.543, E3 +214001.389}
SPL {X  -162.820, Y  +663.189, Z    +0.000, E1   +11.952, E3 +214001.378}
SPL {X  -162.820, Y  +657.986, Z    +0.000, E1   +20.997, E3 +214001.092}
SPL {X  -162.820, Y  +650.033, Z    +0.000, E1   +33.465, E3 +214001.562}
SPL {X  -162.820, Y  +635.632, Z    +0.000, E1   +50.654, E3 +214001.886}
SPL {X  -162.820, Y  +584.142, Z    +0.000, E1   +66.966, E3 +214017.539}
SPL {X  -162.820, Y  +466.182, Z    +0.000, E1   +68.456, E3 +214091.310}
ENDSPLINE

SPLINE
SPL {X  -162.820, Y  +475.083, Z    +0.000, E1   +65.244, E3 +214109.010}
ENDSPLINE

SPLINE
SPL {X  -162.820, Y  +462.171, Z    +0.000, E1   +64.935, E3 +214123.954}
SPL {X  -162.820, Y  +448.581, Z    +0.000, E1   +64.948, E3 +214136.966}
SPL {X  -162.820, Y  +437.579, Z    +0.000, E1   +64.893, E3 +214148.141}
SPL {X  -162.820, Y  +425.248, Z    +0.000, E1   +64.950, E3 +214159.729}
SPL {X  -162.820, Y  +417.868, Z    +0.000, E1   +64.478, E3 +214170.547}
ENDSPLINE

SPLINE
SPL {X  -162.820, Y  +447.149, Z    +0.000, E1   +58.721, E3 +214178.543}
ENDSPLINE

SPLINE
SPL {X  -162.820, Y  +431.862, Z    +0.000, E1   +59.419, E3 +214193.091}
SPL {X  -162.820, Y  +417.107, Z    +0.000, E1   +60.148, E3 +214205.901}
SPL {X  -162.820, Y  +398.797, Z    +0.000, E1   +61.348, E3 +214219.034}
SPL {X  -162.819, Y  +379.881, Z    +0.000, E1   +62.356, E3 +214232.864}
SPL {X  -162.597, Y  +371.985, Z    +0.000, E1   +62.420, E3 +214240.987}
SPL {X  -161.953, Y  +363.716, Z    +0.000, E1   +62.355, E3 +214250.444}
SPL {X  -160.528, Y  +353.277, Z    +0.000, E1   +62.144, E3 +214263.440}
SPL {X  -158.606, Y  +343.697, Z    +0.000, E1   +61.897, E3 +214275.345}
SPL {X  -156.311, Y  +334.925, Z    +0.000, E1   +61.505, E3 +214287.691}
SPL {X  -153.198, Y  +325.358, Z    +0.000, E1   +61.117, E3 +214300.383}
SPL {X  -151.022, Y  +319.651, Z    +0.000, E1   +60.776, E3 +214308.556}
SPL {X  -149.105, Y  +315.094, Z    +0.000, E1   +60.301, E3 +214316.309}
SPL {X  -146.196, Y  +308.826, Z    +0.000, E1   +59.961, E3 +214325.016}
SPL {X  -143.704, Y  +303.952, Z    +0.000, E1   +59.374, E3 +214333.373}
SPL {X  -140.940, Y  +298.976, Z    +0.000, E1   +59.075, E3 +214340.298}
SPL {X  -137.763, Y  +293.715, Z    +0.000, E1   +58.761, E3 +214347.405}
SPL {X  -129.725, Y  +282.103, Z    +0.000, E1   +61.069, E3 +214348.908}
SPL {X  -106.695, Y  +257.510, Z    +0.000, E1   +52.408, E3 +214449.630}
SPL {X  -104.122, Y  +255.325, Z    +0.000, E1   +51.312, E3 +214539.688}
ENDSPLINE

SPLINE
SPL {X  -140.007, Y  +297.383, Z    +0.000, E1   +42.766, E3 +214579.013}
SPL {X  -156.919, Y  +337.064, Z    +0.000, E1   +27.647, E3 +214585.164}
SPL {X  -160.736, Y  +354.534, Z    +0.000, E1   +18.553, E3 +214587.859}
SPL {X  -162.078, Y  +364.978, Z    +0.000, E1   +12.369, E3 +214589.544}
SPL {X  -162.752, Y  +375.778, Z    +0.000, E1    +5.236, E3 +214589.253}
SPL {X  -162.820, Y  +382.443, Z    +0.000, E1    +0.212, E3 +214588.733}
SPL {X  -162.820, Y  +386.214, Z    +0.000, E1    -4.241, E3 +214588.436}
SPL {X  -162.820, Y  +390.506, Z    +0.000, E1   -10.770, E3 +214588.202}
SPL {X  -162.820, Y  +394.643, Z    +0.000, E1   -17.317, E3 +214588.156}
SPL {X  -162.820, Y  +401.515, Z    +0.000, E1   -27.960, E3 +214588.976}
SPL {X  -162.820, Y  +412.105, Z    +0.000, E1   -42.847, E3 +214587.968}
SPL {X  -162.820, Y  +427.270, Z    +0.000, E1   -54.659, E3 +214590.784}
SPL {X  -162.820, Y  +475.967, Z    +0.000, E1   -65.140, E3 +214611.163}
SPL {X  -162.820, Y  +578.686, Z    +0.000, E1   -67.085, E3 +214679.404}
ENDSPLINE

SPLINE
SPL {X  -162.820, Y  +565.364, Z    +0.000, E1   -63.589, E3 +214693.404}
ENDSPLINE

SPLINE
SPL {X  -162.820, Y  +574.608, Z    +0.000, E1   -63.370, E3 +214704.663}
SPL {X  -162.820, Y  +584.314, Z    +0.000, E1   -63.342, E3 +214714.955}
SPL {X  -162.820, Y  +593.857, Z    +0.000, E1   -63.382, E3 +214724.657}
SPL {X  -162.820, Y  +602.272, Z    +0.000, E1   -63.279, E3 +214734.185}
SPL {X  -162.820, Y  +613.309, Z    +0.000, E1   -63.489, E3 +214744.184}
SPL {X  -162.820, Y  +619.956, Z    +0.000, E1   -63.110, E3 +214753.870}
SPL {X  -162.820, Y  +631.846, Z    +0.000, E1   -63.529, E3 +214763.261}
SPL {X  -162.820, Y  +642.772, Z    +0.000, E1   -63.348, E3 +214776.063}
SPL {X  -162.820, Y  +658.642, Z    +0.000, E1   -63.324, E3 +214792.979}
SPL {X  -162.819, Y  +673.983, Z    +0.000, E1   -63.398, E3 +214808.306}
SPL {X  -162.617, Y  +681.634, Z    +0.000, E1   -63.169, E3 +214817.928}
SPL {X  -161.618, Y  +693.246, Z    +0.000, E1   -63.233, E3 +214829.786}
SPL {X  -160.212, Y  +702.527, Z    +0.000, E1   -62.898, E3 +214841.731}
SPL {X  -158.647, Y  +710.128, Z    +0.000, E1   -62.776, E3 +214850.554}
SPL {X  -156.957, Y  +716.799, Z    +0.000, E1   -62.460, E3 +214859.672}
SPL {X  -154.447, Y  +725.041, Z    +0.000, E1   -62.170, E3 +214870.329}
SPL {X  -151.721, Y  +732.586, Z    +0.000, E1   -61.616, E3 +214881.579}
SPL {X  -149.420, Y  +738.185, Z    +0.000, E1   -61.282, E3 +214889.468}
SPL {X  -146.960, Y  +743.593, Z    +0.000, E1   -60.951, E3 +214897.012}
SPL {X  -143.277, Y  +750.844, Z    +0.000, E1   -60.348, E3 +214908.018}
SPL {X  -139.430, Y  +757.582, Z    +0.000, E1   -59.554, E3 +214918.893}
SPL {X  -134.550, Y  +765.187, Z    +0.000, E1   -59.954, E3 +214924.844}
SPL {X  -102.851, Y  +799.722, Z    +0.000, E1   -53.923, E3 +215015.337}
SPL {X  -101.618, Y  +800.716, Z    +0.000, E1   -52.212, E3 +215128.322}
ENDSPLINE

SPLINE
SPL {X  -141.567, Y  +753.931, Z    +0.000, E1   -42.659, E3 +215165.024}
SPL {X  -155.442, Y  +721.958, Z    +0.000, E1   -30.769, E3 +215171.931}
SPL {X  -161.417, Y  +694.832, Z    +0.000, E1   -16.464, E3 +215175.899}
SPL {X  -162.719, Y  +679.228, Z    +0.000, E1    -6.085, E3 +215176.223}
SPL {X  -162.820, Y  +671.750, Z    +0.000, E1    -0.355, E3 +215175.660}
SPL {X  -162.820, Y  +668.525, Z    +0.000, E1    +3.543, E3 +215175.302}
SPL {X  -162.820, Y  +663.189, Z    +0.000, E1   +11.952, E3 +215175.292}
SPL {X  -162.820, Y  +655.445, Z    +0.000, E1   +24.952, E3 +215175.238}
SPL {X  -162.820, Y  +644.088, Z    +0.000, E1   +41.840, E3 +215175.374}
SPL {X  -162.820, Y  +632.645, Z    +0.000, E1   +53.114, E3 +215176.110}
SPL {X  -162.820, Y  +584.142, Z    +0.000, E1   +66.966, E3 +215191.452}
SPL {X  -162.820, Y  +471.906, Z    +0.000, E1   +66.781, E3 +215273.694}
SPL {X  -162.820, Y  +470.218, Z    +0.000, E1   +64.979, E3 +215289.694}
SPL {X  -162.820, Y  +452.619, Z    +0.000, E1   +64.912, E3 +215307.372}
SPL {X  -162.820, Y  +437.579, Z    +0.000, E1   +64.893, E3 +215322.054}
SPL {X  -162.820, Y  +425.248, Z    +0.000, E1   +64.950, E3 +215333.642}
SPL {X  -162.820, Y  +417.868, Z    +0.000, E1   +64.478, E3 +215344.461}
ENDSPLINE

SPLINE
SPL {X  -162.820, Y  +442.889, Z    +0.000, E1   +58.918, E3 +215356.640}
ENDSPLINE

SPLINE
SPL {X  -162.820, Y  +428.091, Z    +0.000, E1   +59.583, E3 +215370.413}
SPL {X  -162.820, Y  +417.107, Z    +0.000, E1   +60.148, E3 +215379.814}
SPL {X  -162.820, Y  +398.797, Z    +0.000, E1   +61.348, E3 +215392.947}
SPL {X  -162.753, Y  +375.814, Z    +0.000, E1   +62.427, E3 +215410.869}
SPL {X  -161.572, Y  +360.382, Z    +0.000, E1   +62.315, E3 +215428.472}
SPL {X  -160.005, Y  +350.357, Z    +0.000, E1   +62.043, E3 +215441.035}
SPL {X  -158.606, Y  +343.697, Z    +0.000, E1   +61.897, E3 +215449.258}
SPL {X  -156.311, Y  +334.925, Z    +0.000, E1   +61.505, E3 +215461.604}
SPL {X  -153.198, Y  +325.358, Z    +0.000, E1   +61.117, E3 +215474.296}
SPL {X  -151.022, Y  +319.651, Z    +0.000, E1   +60.776, E3 +215482.469}
SPL {X  -149.105, Y  +315.094, Z    +0.000, E1   +60.301, E3 +215490.222}
SPL {X  -146.196, Y  +308.826, Z    +0.000, E1   +59.961, E3 +215498.929}
SPL {X  -143.704, Y  +303.952, Z    +0.000, E1   +59.374, E3 +215507.286}
SPL {X  -140.940, Y  +298.976, Z    +0.000, E1   +59.075, E3 +215514.211}
SPL {X  -137.763, Y  +293.715, Z    +0.000, E1   +58.761, E3 +215521.318}
SPL {X  -129.725, Y  +282.103, Z    +0.000, E1   +61.069, E3 +215522.821}
SPL {X  -106.695, Y  +257.510, Z    +0.000, E1   +52.408, E3 +215623.543}
SPL {X  -104.122, Y  +255.325, Z    +0.000, E1   +51.312, E3 +215713.601}
ENDSPLINE

SPLINE
SPL {X  -140.007, Y  +297.383, Z    +0.000, E1   +42.766, E3 +215752.926}
SPL {X  -155.551, Y  +332.393, Z    +0.000, E1   +29.794, E3 +215758.847}
SPL {X  -159.755, Y  +349.054, Z    +0.000, E1   +21.610, E3 +215760.720}
SPL {X  -162.078, Y  +364.978, Z    +0.000, E1   +12.369, E3 +215763.457}
SPL {X  -162.752, Y  +375.778, Z    +0.000, E1    +5.236, E3 +215763.166}
SPL {X  -162.820, Y  +381.939, Z    +0.000, E1    +0.593, E3 +215762.794}
SPL {X  -162.820, Y  +383.993, Z    +0.000, E1    -1.497, E3 +215762.366}
SPL {X  -162.820, Y  +388.628, Z    +0.000, E1    -7.678, E3 +215762.269}
SPL {X  -162.820, Y  +394.643, Z    +0.000, E1   -17.317, E3 +215762.069}
SPL {X  -162.820, Y  +401.515, Z    +0.000, E1   -27.960, E3 +215762.889}
SPL {X  -162.820, Y  +412.105, Z    +0.000, E1   -42.847, E3 +215761.881}
SPL {X  -162.820, Y  +422.796, Z    +0.000, E1   -52.392, E3 +215763.102}
SPL {X  -162.820, Y  +474.423, Z    +0.000, E1   -65.078, E3 +215784.152}
SPL {X  -162.820, Y  +578.686, Z    +0.000, E1   -67.085, E3 +215853.317}
ENDSPLINE

SPLINE
SPL {X  -162.820, Y  +565.364, Z    +0.000, E1   -63.589, E3 +215867.317}
ENDSPLINE

SPLINE
SPL {X  -162.820, Y  +574.608, Z    +0.000, E1   -63.370, E3 +215878.576}
SPL {X  -162.820, Y  +584.314, Z    +0.000, E1   -63.342, E3 +215888.868}
SPL {X  -162.820, Y  +593.857, Z    +0.000, E1   -63.382, E3 +215898.570}
SPL {X  -162.820, Y  +602.272, Z    +0.000, E1   -63.279, E3 +215908.099}
SPL {X  -162.820, Y  +613.309, Z    +0.000, E1   -63.489, E3 +215918.097}
SPL {X  -162.820, Y  +619.956, Z    +0.000, E1   -63.110, E3 +215927.783}
SPL {X  -162.820, Y  +631.846, Z    +0.000, E1   -63.529, E3 +215937.174}
SPL {X  -162.820, Y  +642.772, Z    +0.000, E1   -63.348, E3 +215949.976}
SPL {X  -162.820, Y  +658.642, Z    +0.000, E1   -63.324, E3 +215966.892}
SPL {X  -162.819, Y  +673.983, Z    +0.000, E1   -63.398, E3 +215982.219}
SPL {X  -162.399, Y  +685.202, Z    +0.000, E1   -63.235, E3 +215995.213}
SPL {X  -161.289, Y  +695.772, Z    +0.000, E1   -63.167, E3 +216006.663}
SPL {X  -160.212, Y  +702.527, Z    +0.000, E1   -62.898, E3 +216015.644}
SPL {X  -158.647, Y  +710.128, Z    +0.000, E1   -62.776, E3 +216024.467}
SPL {X  -156.957, Y  +716.799, Z    +0.000, E1   -62.460, E3 +216033.585}
SPL {X  -154.447, Y  +725.041, Z    +0.000, E1   -62.170, E3 +216044.242}
SPL {X  -151.721, Y  +732.586, Z    +0.000, E1   -61.616, E3 +216055.492}
SPL {X  -149.420, Y  +738.185, Z    +0.000, E1   -61.282, E3 +216063.381}
SPL {X  -146.960, Y  +743.593, Z    +0.000, E1   -60.951, E3 +216070.925}
SPL {X  -143.277, Y  +750.844, Z    +0.000, E1   -60.348, E3 +216081.931}
SPL {X  -139.430, Y  +757.582, Z    +0.000, E1   -59.554, E3 +216092.806}
SPL {X  -134.550, Y  +765.187, Z    +0.000, E1   -59.954, E3 +216098.757}
SPL {X  -100.103, Y  +801.912, Z    +0.000, E1   -53.794, E3 +216196.807}
ENDSPLINE

SPLINE
SPL {X  -112.938, Y  +790.784, Z    +0.000, E1   -51.983, E3 +216332.329}
SPL {X  -141.567, Y  +753.931, Z    +0.000, E1   -42.659, E3 +216338.937}
SPL {X  -155.442, Y  +721.958, Z    +0.000, E1   -30.769, E3 +216345.844}
SPL {X  -161.417, Y  +694.832, Z    +0.000, E1   -16.464, E3 +216349.812}
SPL {X  -162.719, Y  +679.228, Z    +0.000, E1    -6.085, E3 +216350.136}
SPL {X  -162.820, Y  +673.638, Z    +0.000, E1    -1.806, E3 +216349.926}
SPL {X  -162.820, Y  +670.948, Z    +0.000, E1    +0.412, E3 +216349.451}
SPL {X  -162.820, Y  +667.375, Z    +0.000, E1    +5.386, E3 +216349.140}
SPL {X  -162.820, Y  +663.189, Z    +0.000, E1   +11.952, E3 +216349.205}
SPL {X  -162.820, Y  +655.445, Z    +0.000, E1   +24.952, E3 +216349.151}
SPL {X  -162.820, Y  +644.088, Z    +0.000, E1   +41.840, E3 +216349.287}
SPL {X  -162.820, Y  +632.645, Z    +0.000, E1   +53.114, E3 +216350.023}
SPL {X  -162.820, Y  +584.142, Z    +0.000, E1   +66.966, E3 +216365.365}
SPL {X  -162.820, Y  +471.906, Z    +0.000, E1   +66.781, E3 +216447.607}
SPL {X  -162.820, Y  +470.218, Z    +0.000, E1   +64.979, E3 +216463.607}
SPL {X  -162.820, Y  +452.619, Z    +0.000, E1   +64.912, E3 +216481.285}
SPL {X  -162.820, Y  +437.579, Z    +0.000, E1   +64.893, E3 +216495.967}
SPL {X  -162.820, Y  +425.248, Z    +0.000, E1   +64.950, E3 +216507.555}
SPL {X  -162.820, Y  +417.868, Z    +0.000, E1   +64.478, E3 +216518.374}
ENDSPLINE

SPLINE
SPL {X  -162.820, Y  +447.149, Z    +0.000, E1   +58.721, E3 +216526.369}
ENDSPLINE

SPLINE
SPL {X  -162.820, Y  +431.862, Z    +0.000, E1   +59.419, E3 +216540.917}
SPL {X  -162.820, Y  +417.107, Z    +0.000, E1   +60.148, E3 +216553.727}
SPL {X  -162.820, Y  +398.797, Z    +0.000, E1   +61.348, E3 +216566.860}
SPL {X  -162.753, Y  +375.814, Z    +0.000, E1   +62.427, E3 +216584.782}
SPL {X  -161.953, Y  +363.716, Z    +0.000, E1   +62.355, E3 +216598.270}
SPL {X  -160.528, Y  +353.277, Z    +0.000, E1   +62.144, E3 +216611.267}
SPL {X  -157.973, Y  +341.066, Z    +0.000, E1   +61.800, E3 +216626.865}
SPL {X  -155.627, Y  +332.640, Z    +0.000, E1   +61.354, E3 +216638.779}
SPL {X  -153.198, Y  +325.358, Z    +0.000, E1   +61.117, E3 +216648.209}
SPL {X  -151.022, Y  +319.651, Z    +0.000, E1   +60.776, E3 +216656.382}
SPL {X  -149.105, Y  +315.094, Z    +0.000, E1   +60.301, E3 +216664.135}
SPL {X  -146.196, Y  +308.826, Z    +0.000, E1   +59.961, E3 +216672.842}
SPL {X  -143.704, Y  +303.952, Z    +0.000, E1   +59.374, E3 +216681.199}
SPL {X  -140.940, Y  +298.976, Z    +0.000, E1   +59.075, E3 +216688.124}
SPL {X  -137.763, Y  +293.715, Z    +0.000, E1   +58.761, E3 +216695.231}
SPL {X  -129.725, Y  +282.103, Z    +0.000, E1   +61.069, E3 +216696.734}
SPL {X  -106.695, Y  +257.510, Z    +0.000, E1   +52.408, E3 +216797.456}
SPL {X  -104.122, Y  +255.325, Z    +0.000, E1   +51.312, E3 +216887.514}
ENDSPLINE

SPLINE
SPL {X  -140.007, Y  +297.383, Z    +0.000, E1   +42.766, E3 +216926.839}
SPL {X  -156.919, Y  +337.064, Z    +0.000, E1   +27.647, E3 +216932.990}
SPL {X  -161.737, Y  +361.753, Z    +0.000, E1   +14.421, E3 +216936.887}
SPL {X  -162.752, Y  +375.778, Z    +0.000, E1    +5.236, E3 +216937.079}
SPL {X  -162.820, Y  +382.443, Z    +0.000, E1    +0.212, E3 +216936.559}
SPL {X  -162.820, Y  +386.214, Z    +0.000, E1    -4.241, E3 +216936.262}
SPL {X  -162.820, Y  +390.506, Z    +0.000, E1   -10.770, E3 +216936.028}
SPL {X  -162.820, Y  +394.643, Z    +0.000, E1   -17.317, E3 +216935.982}
SPL {X  -162.820, Y  +401.515, Z    +0.000, E1   -27.960, E3 +216936.802}
SPL {X  -162.820, Y  +412.105, Z    +0.000, E1   -42.847, E3 +216935.794}
SPL {X  -162.820, Y  +422.796, Z    +0.000, E1   -52.392, E3 +216937.015}
SPL {X  -162.820, Y  +474.423, Z    +0.000, E1   -65.078, E3 +216958.066}
SPL {X  -162.820, Y  +578.686, Z    +0.000, E1   -67.085, E3 +217027.230}
ENDSPLINE

SPLINE
SPL {X  -162.820, Y  +565.364, Z    +0.000, E1   -63.589, E3 +217041.230}
ENDSPLINE

SPLINE
SPL {X  -162.820, Y  +574.608, Z    +0.000, E1   -63.370, E3 +217052.489}
SPL {X  -162.820, Y  +584.314, Z    +0.000, E1   -63.342, E3 +217062.781}
SPL {X  -162.820, Y  +593.857, Z    +0.000, E1   -63.382, E3 +217072.484}
SPL {X  -162.820, Y  +602.272, Z    +0.000, E1   -63.279, E3 +217082.012}
SPL {X  -162.820, Y  +613.309, Z    +0.000, E1   -63.489, E3 +217092.010}
SPL {X  -162.820, Y  +627.013, Z    +0.000, E1   -63.389, E3 +217107.231}
SPL {X  -162.820, Y  +642.772, Z    +0.000, E1   -63.348, E3 +217123.890}
SPL {X  -162.820, Y  +658.642, Z    +0.000, E1   -63.324, E3 +217140.805}
SPL {X  -162.819, Y  +673.983, Z    +0.000, E1   -63.398, E3 +217156.132}
SPL {X  -162.617, Y  +681.634, Z    +0.000, E1   -63.169, E3 +217165.755}
SPL {X  -161.618, Y  +693.246, Z    +0.000, E1   -63.233, E3 +217177.612}
SPL {X  -160.212, Y  +702.527, Z    +0.000, E1   -62.898, E3 +217189.557}
SPL {X  -158.647, Y  +710.128, Z    +0.000, E1   -62.776, E3 +217198.380}
SPL {X  -156.957, Y  +716.799, Z    +0.000, E1   -62.460, E3 +217207.498}
SPL {X  -155.130, Y  +722.947, Z    +0.000, E1   -62.207, E3 +217215.610}
SPL {X  -152.287, Y  +731.112, Z    +0.000, E1   -61.798, E3 +217226.885}
SPL {X  -149.420, Y  +738.185, Z    +0.000, E1   -61.282, E3 +217237.294}
SPL {X  -146.033, Y  +745.504, Z    +0.000, E1   -60.844, E3 +217247.561}
SPL {X  -142.518, Y  +752.234, Z    +0.000, E1   -60.144, E3 +217258.187}
SPL {X  -139.430, Y  +757.582, Z    +0.000, E1   -59.554, E3 +217266.719}
SPL {X  -134.550, Y  +765.187, Z    +0.000, E1   -59.954, E3 +217272.670}
SPL {X  -100.103, Y  +801.912, Z    +0.000, E1   -53.794, E3 +217370.720}
ENDSPLINE

SPLINE
SPL {X  -112.938, Y  +790.784, Z    +0.000, E1   -51.983, E3 +217506.242}
SPL {X  -141.567, Y  +753.931, Z    +0.000, E1   -42.659, E3 +217512.850}
SPL {X  -155.442, Y  +721.958, Z    +0.000, E1   -30.769, E3 +217519.757}
SPL {X  -161.417, Y  +694.832, Z    +0.000, E1   -16.464, E3 +217523.725}
SPL {X  -162.719, Y  +679.228, Z    +0.000, E1    -6.085, E3 +217524.049}
SPL {X  -162.820, Y  +673.638, Z    +0.000, E1    -1.806, E3 +217523.839}
SPL {X  -162.820, Y  +670.948, Z    +0.000, E1    +0.412, E3 +217523.364}
SPL {X  -162.820, Y  +667.375, Z    +0.000, E1    +5.386, E3 +217523.053}
SPL {X  -162.820, Y  +663.189, Z    +0.000, E1   +11.952, E3 +217523.118}
SPL {X  -162.820, Y  +655.445, Z    +0.000, E1   +24.952, E3 +217523.064}
SPL {X  -162.820, Y  +644.088, Z    +0.000, E1   +41.840, E3 +217523.200}
SPL {X  -162.820, Y  +632.645, Z    +0.000, E1   +53.114, E3 +217523.936}
SPL {X  -162.820, Y  +584.142, Z    +0.000, E1   +66.966, E3 +217539.278}
SPL {X  -162.820, Y  +466.182, Z    +0.000, E1   +68.456, E3 +217613.049}
ENDSPLINE

SPLINE
SPL {X  -162.820, Y  +475.083, Z    +0.000, E1   +65.244, E3 +217630.749}
ENDSPLINE

SPLINE
SPL {X  -162.820, Y  +465.389, Z    +0.000, E1   +65.015, E3 +217641.766}
SPL {X  -162.820, Y  +452.619, Z    +0.000, E1   +64.912, E3 +217655.198}
SPL {X  -162.820, Y  +437.579, Z    +0.000, E1   +64.893, E3 +217669.880}
SPL {X  -162.820, Y  +425.248, Z    +0.000, E1   +64.950, E3 +217681.468}
SPL {X  -162.820, Y  +417.868, Z    +0.000, E1   +64.478, E3 +217692.287}
ENDSPLINE

SPLINE
SPL {X  -162.820, Y  +442.889, Z    +0.000, E1   +58.918, E3 +217704.467}
ENDSPLINE

SPLINE
SPL {X  -162.820, Y  +428.091, Z    +0.000, E1   +59.583, E3 +217718.239}
SPL {X  -162.820, Y  +417.107, Z    +0.000, E1   +60.148, E3 +217727.640}
SPL {X  -162.820, Y  +398.797, Z    +0.000, E1   +61.348, E3 +217740.773}
SPL {X  -162.819, Y  +379.881, Z    +0.000, E1   +62.356, E3 +217754.603}
SPL {X  -162.597, Y  +371.985, Z    +0.000, E1   +62.420, E3 +217762.726}
SPL {X  -161.953, Y  +363.716, Z    +0.000, E1   +62.355, E3 +217772.184}
SPL {X  -160.528, Y  +353.277, Z    +0.000, E1   +62.144, E3 +217785.180}
SPL {X  -158.606, Y  +343.697, Z    +0.000, E1   +61.897, E3 +217797.084}
SPL {X  -156.311, Y  +334.925, Z    +0.000, E1   +61.505, E3 +217809.430}
SPL {X  -153.198, Y  +325.358, Z    +0.000, E1   +61.117, E3 +217822.122}
SPL {X  -151.022, Y  +319.651, Z    +0.000, E1   +60.776, E3 +217830.295}
SPL {X  -149.105, Y  +315.094, Z    +0.000, E1   +60.301, E3 +217838.048}
SPL {X  -146.196, Y  +308.826, Z    +0.000, E1   +59.961, E3 +217846.755}
SPL {X  -143.704, Y  +303.952, Z    +0.000, E1   +59.374, E3 +217855.112}
SPL {X  -140.940, Y  +298.976, Z    +0.000, E1   +59.075, E3 +217862.037}
SPL {X  -137.763, Y  +293.715, Z    +0.000, E1   +58.761, E3 +217869.144}
SPL {X  -129.725, Y  +282.103, Z    +0.000, E1   +61.069, E3 +217870.647}
SPL {X  -106.695, Y  +257.510, Z    +0.000, E1   +52.408, E3 +217971.369}
SPL {X  -104.122, Y  +255.325, Z    +0.000, E1   +51.312, E3 +218061.427}
ENDSPLINE

SPLINE
SPL {X  -140.007, Y  +297.383, Z    +0.000, E1   +42.766, E3 +218100.752}
SPL {X  -156.919, Y  +337.064, Z    +0.000, E1   +27.647, E3 +218106.903}
SPL {X  -160.736, Y  +354.534, Z    +0.000, E1   +18.553, E3 +218109.598}
SPL {X  -162.078, Y  +364.978, Z    +0.000, E1   +12.369, E3 +218111.283}
SPL {X  -162.656, Y  +373.196, Z    +0.000, E1    +6.960, E3 +218110.779}
SPL {X  -162.819, Y  +379.805, Z    +0.000, E1    +2.285, E3 +218110.903}
SPL {X  -162.820, Y  +382.398, Z    +0.000, E1    +0.126, E3 +218110.562}
SPL {X  -162.820, Y  +383.993, Z    +0.000, E1    -1.497, E3 +218110.192}
SPL {X  -162.820, Y  +387.367, Z    +0.000, E1    -6.003, E3 +218110.198}
SPL {X  -162.820, Y  +390.506, Z    +0.000, E1   -10.770, E3 +218109.941}
SPL {X  -162.820, Y  +394.643, Z    +0.000, E1   -17.317, E3 +218109.895}
SPL {X  -162.820, Y  +401.515, Z    +0.000, E1   -27.960, E3 +218110.715}
SPL {X  -162.820, Y  +412.105, Z    +0.000, E1   -42.847, E3 +218109.707}
SPL {X  -162.820, Y  +422.796, Z    +0.000, E1   -52.392, E3 +218110.928}
SPL {X  -162.820, Y  +474.423, Z    +0.000, E1   -65.078, E3 +218131.979}
SPL {X  -162.820, Y  +578.686, Z    +0.000, E1   -67.085, E3 +218201.143}
ENDSPLINE

SPLINE
SPL {X  -162.820, Y  +565.364, Z    +0.000, E1   -63.589, E3 +218215.143}
ENDSPLINE

SPLINE
SPL {X  -162.820, Y  +574.608, Z    +0.000, E1   -63.370, E3 +218226.402}
SPL {X  -162.820, Y  +584.314, Z    +0.000, E1   -63.342, E3 +218236.694}
SPL {X  -162.820, Y  +593.857, Z    +0.000, E1   -63.382, E3 +218246.397}
SPL {X  -162.820, Y  +602.272, Z    +0.000, E1   -63.279, E3 +218255.925}
SPL {X  -162.820, Y  +613.309, Z    +0.000, E1   -63.489, E3 +218265.923}
SPL {X  -162.820, Y  +619.956, Z    +0.000, E1   -63.110, E3 +218275.610}
SPL {X  -162.820, Y  +634.513, Z    +0.000, E1   -63.471, E3 +218288.376}
SPL {X  -162.820, Y  +648.936, Z    +0.000, E1   -63.278, E3 +218304.831}
SPL {X  -162.820, Y  +662.662, Z    +0.000, E1   -63.383, E3 +218318.323}
SPL {X  -162.819, Y  +673.983, Z    +0.000, E1   -63.398, E3 +218330.045}
SPL {X  -162.399, Y  +685.202, Z    +0.000, E1   -63.235, E3 +218343.039}
SPL {X  -161.289, Y  +695.772, Z    +0.000, E1   -63.167, E3 +218354.489}
SPL {X  -160.212, Y  +702.527, Z    +0.000, E1   -62.898, E3 +218363.470}
SPL {X  -158.647, Y  +710.128, Z    +0.000, E1   -62.776, E3 +218372.293}
SPL {X  -156.957, Y  +716.799, Z    +0.000, E1   -62.460, E3 +218381.411}
SPL {X  -154.447, Y  +725.041, Z    +0.000, E1   -62.170, E3 +218392.068}
SPL {X  -151.721, Y  +732.586, Z    +0.000, E1   -61.616, E3 +218403.318}
SPL {X  -149.420, Y  +738.185, Z    +0.000, E1   -61.282, E3 +218411.207}
SPL {X  -146.960, Y  +743.593, Z    +0.000, E1   -60.951, E3 +218418.751}
SPL {X  -143.277, Y  +750.844, Z    +0.000, E1   -60.348, E3 +218429.757}
SPL {X  -139.430, Y  +757.582, Z    +0.000, E1   -59.554, E3 +218440.632}
SPL {X  -134.550, Y  +765.187, Z    +0.000, E1   -59.954, E3 +218446.583}
SPL {X  -100.103, Y  +801.912, Z    +0.000, E1   -53.794, E3 +218544.633}
ENDSPLINE

SPLINE
SPL {X  -112.938, Y  +790.784, Z    +0.000, E1   -51.983, E3 +218680.155}
SPL {X  -145.058, Y  +747.450, Z    +0.000, E1   -40.634, E3 +218688.265}
SPL {X  -158.857, Y  +709.206, Z    +0.000, E1   -24.633, E3 +218696.234}
SPL {X  -161.919, Y  +690.607, Z    +0.000, E1   -13.733, E3 +218697.714}
SPL {X  -162.719, Y  +679.228, Z    +0.000, E1    -6.085, E3 +218697.962}
SPL {X  -162.820, Y  +671.750, Z    +0.000, E1    -0.355, E3 +218697.399}
SPL {X  -162.820, Y  +669.853, Z    +0.000, E1    +1.938, E3 +218697.129}
SPL {X  -162.820, Y  +667.375, Z    +0.000, E1    +5.386, E3 +218696.966}
SPL {X  -162.820, Y  +663.189, Z    +0.000, E1   +11.952, E3 +218697.031}
SPL {X  -162.820, Y  +655.445, Z    +0.000, E1   +24.952, E3 +218696.977}
SPL {X  -162.820, Y  +644.088, Z    +0.000, E1   +41.840, E3 +218697.113}
SPL {X  -162.820, Y  +632.645, Z    +0.000, E1   +53.114, E3 +218697.849}
SPL {X  -162.820, Y  +584.142, Z    +0.000, E1   +66.966, E3 +218713.191}
SPL {X  -162.820, Y  +471.906, Z    +0.000, E1   +66.781, E3 +218795.433}
SPL {X  -162.820, Y  +470.218, Z    +0.000, E1   +64.979, E3 +218811.433}
SPL {X  -162.820, Y  +452.619, Z    +0.000, E1   +64.912, E3 +218829.111}
SPL {X  -162.820, Y  +437.579, Z    +0.000, E1   +64.893, E3 +218843.793}
SPL {X  -162.820, Y  +425.248, Z    +0.000, E1   +64.950, E3 +218855.381}
SPL {X  -162.820, Y  +417.868, Z    +0.000, E1   +64.478, E3 +218866.200}
ENDSPLINE

SPLINE
SPL {X  -162.820, Y  +442.889, Z    +0.000, E1   +58.918, E3 +218878.380}
ENDSPLINE

